Encoder_Extendido := gEncoder_AbsolutoExtendido;
Encoder_Parada := gEncoder_OperativaB;
TeachingOperativaB := gEncoder_Absoluto - 40000;            //----- Valor que permite el inicio del teaching del encoder de parada -----//
Encoder_Extendido_OFFSET := 150;							//----- Valor para los casos de anomalia en que no detectamos inductivo de brazo extendido -----//
Encoder_Recogido_OFFSET := 150;								//----- Valor para los casos de anomalia en que no detectamos inductivo de brazo recogido -----//

Encoder_Parada_OFFSET := 200;								//----- Valor de OFFSET para la parada del brazo por encoder -----//

C40.NumID:=1;
C40.MatrizID[1]:=65;
C41.RespuestasTotales[1]:=16#1F;        					//----- Tiene que recibir informacion de 5 PDOs -----//

//-------------------------------------------------------------------------------------------//
//----------------------------Definicion temporizacion inicial-------------------------------//
//-------------------------------------------------------------------------------------------//
SEGUNDOS_ENCENDIDO := 10;
TIEMPO_CICLO_DESEADO := 15000;

//-------------------------------------------------------------------------------------------//
//----------------------------------------Anomalias------------------------------------------//
//-------------------------------------------------------------------------------------------//
//TIPO_ANOMALIA[0]  := 3;	
//----- Anomalias supervisor -----//
TIPO_ANOMALIA[1]  := 3;		
TIPO_ANOMALIA[2]  := 1;	

//----- Anomalias imágenes -----//
TIPO_ANOMALIA[3]  := 3;		
TIPO_ANOMALIA[4]  := 4;		
TIPO_ANOMALIA[5]  := 3;		
TIPO_ANOMALIA[6]  := 3;		
TIPO_ANOMALIA[7]  := 3;	
TIPO_ANOMALIA[8]  := 3;		
TIPO_ANOMALIA[9]  := 3;	

//----- Anomalías estados -----//
TIPO_ANOMALIA[10] := 1;		
TIPO_ANOMALIA[11] := 2;		
TIPO_ANOMALIA[12] := 2;		
TIPO_ANOMALIA[13] := 2;		
TIPO_ANOMALIA[14] := 2;		
TIPO_ANOMALIA[15] := 3;
TIPO_ANOMALIA[16] := 2;		
TIPO_ANOMALIA[17] := 0;	

//----- Anomalías secuencia carga -----//
TIPO_ANOMALIA[18] := 4;		
TIPO_ANOMALIA[19] := 1;		
TIPO_ANOMALIA[20] := 3;		
TIPO_ANOMALIA[21] := 2;		
TIPO_ANOMALIA[22] := 3;		
TIPO_ANOMALIA[23] := 3; 
TIPO_ANOMALIA[24] := 3;		
//TIPO_ANOMALIA[25] := 2;	

//----- Anomalías extensión -----//
TIPO_ANOMALIA[26] := 2;		 
TIPO_ANOMALIA[27] := 3;		
TIPO_ANOMALIA[28] := 2;		
TIPO_ANOMALIA[29] := 2;		
TIPO_ANOMALIA[30] := 2;		
TIPO_ANOMALIA[31] := 2; 

//----- Anomalías elevación -----//
TIPO_ANOMALIA[32] := 3;		
TIPO_ANOMALIA[33] := 2;		
TIPO_ANOMALIA[34] := 4;		
(*TIPO_ANOMALIA[35] := 2;		
TIPO_ANOMALIA[36] := 2;		
TIPO_ANOMALIA[37] := 2;		
TIPO_ANOMALIA[38] := 2;		
TIPO_ANOMALIA[39] := 2; *)

END_PROGRAM

// StandardPLC/Application/CÓDIGO/SUPERVISOR
PROGRAM SUPERVISOR
VAR CONSTANT
	TOTALANOMALIAS 			:INT := 39;
END_VAR
VAR
	estadoAnomalias	  		:ARRAY[0..TOTALANOMALIAS] OF BYTE;
	anomaliasEntrada 		:ARRAY[0..TOTALANOMALIAS] OF BOOL;
	rearme 					:BOOL;
	estadoManual 			:BOOL;
	A_EstadoReposo 			:BOOL;

	mensajeAnomalia 		:BYTE;
	controlEstados 			:BYTE;

	(*Auxiliares*)
	i 						:INT;
	j 						:INT;
END_VAR
VAR_OUTPUT
END_VAR

(*//////////////////////////////////////////////////////////////////////////////////////////////////////////////////////////////////////////////////////////////////////////////////////////////////////////////////////////////////////////////////
SUPERVISOR (PRG)                     

Description:	Las anomalias son administradas en este modulo.
				Existen 4 estados distintos de anomalia (variable estadoAnomalias):
					0: Activa
					1: desactivada
					2: pausa
					3: seguro
				Para cada anomalia, tenemos 5 valores de severidad:
					0: Advertencia autorearmable
					1: Advertencia rearmable
					2: Severa (E-Frame a estado seguro)
					3: Crítica (rearmable con seta)
					4: Fatal (no rearmable)
				
				Cuando no tenemos anomalia, el valor es 1. Siempre que es detectada una anomalia, el valor es cambiado para 0

////////////////////////////////////////////////////////////////////////////////////////////////////////////////////////////////////////////////////////////////////////////////////////////////////////////////////////////////////////////////////*)

//-------------------------------------------------------------------------------------------//
//-------------------------Hacer reset a la variable estadoAnomalias-------------------------//
//-------------------------------------------------------------------------------------------//
IF PrimerCiclo THEN
	TIPO_ANOMALIA[1] := 3;									//----- Anomalía cadena seguridad -----//
	FOR i:=0 TO TOTALANOMALIAS DO 
		estadoAnomalias[i] := 1;            				//----- Para todas las anomalias contempladas en la PARAMETRIZACION, el estado de anomalia es iniciado como anomalia desactivada -----//
	END_FOR;
END_IF;

IF gFinEncendido THEN
	
	anomaliasEntrada 	:= gSupE_AnomaliasEntrada;
	rearme 				:= gEntradasPLC.BotonRearme;       
	estadoManual 		:= (gEstadoEframe=Manual) OR (gEstadoEframe=Automatico); 
	A_EstadoReposo 		:= ((gEstadoCarga=cargado) OR (gEstadoCarga=descargado));
	
	//----------------------- estadoAnomalias para la cadena de seguridad -------------------------//
	IF (NOT anomaliasEntrada[1]) THEN
		estadoAnomalias[1] := 0;
	ELSIF ( (estadoAnomalias[1]=0) AND anomaliasEntrada[1] ) THEN
		estadoAnomalias[1] := 3;
	ELSIF ( (estadoAnomalias[1]=3) AND rearme ) THEN    			//----- Si tenemos anomalia en la seta -----//
		IF A_EstadoReposo THEN      								//----- y tenemos en E-Frame cargado o descargado -----//
			estadoAnomalias[1] := 1;     							//----- pasamos el estado de la anomalia como siendo una advertencia autorearmable activa -----//
		ELSE 
			estadoAnomalias[1] := 2;     							//----- si no , tenemos una anomalia severa -----//
		END_IF;
	ELSIF ( (estadoAnomalias[1]=2) AND estadoManual ) THEN     		//----- tenemos una anomalia severa en la cadena de seguridad y estamos en modo manual -----//
		estadoAnomalias[1] := 1;                               		//----- pasamos el estado de la anomalia para una advertencia autorearmable activa -----//
	END_IF;

	//----------------------------------Cambiar estadoAnomalias----------------------------------//
	FOR i:=1 TO (TOTALANOMALIAS-1) DO
		CASE TIPO_ANOMALIA[i] OF
			0: // Advertencia autorearmable. Cuando desaparece origen anomalía. 0:ACTIVA, 1:DESACTIVADA
				estadoAnomalias[i] := BOOL_TO_BYTE(anomaliasEntrada[i]);
			1: // Advertencia rearmable  . Limpiamos anomalía con REARMAR. 0:ACTIVA, 1:DESACTIVADA
				IF (NOT anomaliasEntrada[i]) THEN     				//----- Si tenemos una anomalia, cambiamos su estado para ACTIVO -----//
					estadoAnomalias[i] := 0;
				END_IF;
				IF ( rearme ) THEN    								//----- Así que pulsemos rearme, desactivamos la variable de anomalia -----//
					estadoAnomalias[i] := 1; 
				END_IF;
			2: // Severa - a estado seguro. Permite pausar anomalía con REARMAR, pero desaparece cuando entramos en degradado/manual para corrección.
			    // 0:ACTIVA, 1:DESACTIVADA, 2:PAUSA
				IF ( (estadoAnomalias[i]=1) AND (NOT anomaliasEntrada[i]) ) THEN     //----- Si la variable de anomalia esta desactiva y tenemos una anomalia, pasamos la variable para el estado ACTIVO -----//
					estadoAnomalias[i] := 0;
				ELSIF ( (estadoAnomalias[i]=0) AND rearme ) THEN     //----- Si la variable de anomalia esta en estado activo y pulsamos rearme, ponemos su estado como sendo PAUSA -----//
					estadoAnomalias[i] := 2;
				ELSIF ( ((estadoAnomalias[i]=2) OR (estadoAnomalias[i]=0)) AND rearme ) THEN    //----- Si tenemos el estado de la variable como PAUSA o ACTIVA y cambiamos a modo manual, quitamos anomalia -----//
					estadoAnomalias[i] := 1;
				END_IF;
			3: // Crítica - rearmable con seta . Requieren reset por parte de cadena de seguridad. 0:ACTIVA, 1:DESACTIVADA
				gSalidasPLC.LuzBotonRearme := TOF_Rearme.Q;
				IF rearme THEN        //----- Si cargamos el boton rearme, quitamos la anomalia. Si no, si continuamos con anomalia, la variable estadoAnomalias continua con anomalia activa -----//
					estadoAnomalias[i] := 1;
					gSalidasPLC.LuzBotonRearme := FALSE;
				ELSIF (NOT anomaliasEntrada[i]) THEN
					estadoAnomalias[i] := 0;
				END_IF;
			4: // Fatal - no rearmable. Podemos pausar con cadena de seguridad, pero no se rearmarán. 0:ACTIVA, 1:DESACTIVADA, 2:PAUSA
				IF ( (estadoAnomalias[i]=1) AND (NOT anomaliasEntrada[i]) ) THEN    //----- Si la variable esta DESACTIVA y tenemos una anomalia, cambiamos el estado de la variable para ACTIVA -----//
					estadoAnomalias[i] := 0;
				ELSIF ( (estadoAnomalias[i]=0) AND rearme ) THEN     //----- Si la variables de las anomalias esta ACTIVA y pulsamos rearme, cambiamos su estado para PAUSA	-----//
					estadoAnomalias[i] := 2;
				END_IF;
		END_CASE;
	END_FOR;

	//----- Si tenemos anomalias en extension, reset respectivo módulo control -----//
	gSupS_ResetExtension :=0;

	FOR i:=26 TO 31 DO					
		IF (anomaliasEntrada[i]=0) AND (NOT LASER_AUX) THEN     //----- Si tenemos alguna anomalia -----//
			gSupS_ResetExtension :=1;       					//----- Pasa la variable a 1. Desencadea anomalia en el brazo -----//
			EXIT; 
		END_IF; 	
	END_FOR;
	
	controlEstados 		:= 0;
	mensajeAnomalia 	:= 0;
	
	//----- De acuerdo con el tipo de anomalia que tenemos, vamos escribir la variable mensajeAnomalia para enviar al AGV -----//
	IF ( estadoAnomalias[1]=0 ) THEN   				//----- Anomalia cadena de seguridad -----//
		mensajeAnomalia := 1;	
		controlEstados := 6;
	ELSIF ( estadoAnomalias[1]=3 ) THEN     		//----- Cadena de seguridad en estado seguro -----//
		mensajeAnomalia := 2;	
		controlEstados := 4;
	ELSE
		FOR j:=4 TO 0 BY (-1) DO                   //----- De más a menos severidad -----//
			FOR i:=3 TO (TOTALANOMALIAS-1) DO      //----- Todas las anomalías -----//
				IF ( TIPO_ANOMALIA[i]=j) AND (estadoAnomalias[i]<>1 ) THEN      //----- Si para i tenemos la anomalia j y la variable de anomalia esta en un caso distinto de DESACTIVO -----//
					mensajeAnomalia := INT_TO_BYTE(i);
					CASE j OF
						0: controlEstados := 1;
						1: controlEstados := 5;
						2: 	IF estadoAnomalias[i]=0 THEN 
								controlEstados := 3; 
							ELSE controlEstados := 2;    //----- Si hemos quitado la seta, entra en el seguiente estado de anomalia que es el 3 (necesario llevar E-Frame a posicion inicial) -----//
								mensajeAnomalia := 3; 
							END_IF;
						3: 	IF estadoAnomalias[i]=0 THEN 
								controlEstados := 6; 
							ELSE 
								controlEstados := 2; 
								mensajeAnomalia := 2; //3
							END_IF;
						4: 	IF estadoAnomalias[i]=0 THEN 
								controlEstados := 6; 
							ELSE 
								controlEstados := 4; 
							END_IF;
					END_CASE;
					EXIT;
				END_IF;
			END_FOR;

			IF ( mensajeAnomalia<>0 ) THEN		//----- Si tenemos valor en la variable mensajeAnomalia, tenemos anomalia -----//
				EXIT;
			END_IF;

		END_FOR;
	END_IF;

	gSupS_MensajeAnom 		:= mensajeAnomalia;
	gSupS_ControlEstados 	:= controlEstados;
END_IF;

END_PROGRAM

// StandardPLC/Application/CÓDIGO/ESTADOS
	PROGRAM ESTADOS
VAR
	OrdenDegradado			:BOOL;
	OrdenManual				:BOOL;
	OrdenAuto				:BOOL;
	FrenteAestacion			:BOOL;

	TON_SalirManual			:TON;
	
	Tempo_Actual 			:TIME;
	RetenerEstado			:EstadoEframe;
	CondicionReinicio		:BOOL;
	EstadoAnomaliaA			:BYTE;

	AnomaliaIndeterminado 	:BOOL;
	TON_Posicionado 		:TON;
	AnomaliaPartida 		:BOOL;
	TON_AnomaliaReinicio	:TON;
	AnomaliaReinicio		:BOOL;
END_VAR
VAR_OUTPUT
END_VAR

(*//////////////////////////////////////////////////////////////////////////////////////////////////////////////////////////////////////////////////////////////////////////////////////////////////////////////////////////////////////////////////
ESTADOS (PRG)                     

Description:  Máquina estados principal e-frame. Tenemos 7 estados:

				Identificar 	-> Condiciones arranque. Identifica estado seguro.
				Reposo			-> Brazo retraído, sin orden de carga o descarga.
				Automatico		-> E-Frame ejecutando operativa em modo automatico.
				Degradado		-> Control del brazo con auxilio de un taladro. Salidas del PLC desactivas.
				Manual			-> Control del E-Frame por botones (movimiento del brazo y movimiento de las levas). 
								En este modo, no tenemos anomalias.
				Reinicio		-> Estado utilizado para cuando salimos del modo manual o degradado.
				Anomalía		-> Fueron detetadas anomalias en el funcionamiento.

/////////////////////////////////////////////////////////////////////////////////////////////////////////////////////////////////////////////////////////////////////////////////////////////////////////////////////////////////////////////////////*)

IF gFinEncendido THEN
	//-------------------------------------------------------------------------------------------//
	//-----------CASE para el control del estado de la carga cuando iniciamos E-Frame------------//
	//-------------------------------------------------------------------------------------------//
	IF (gCargaOPT = indeterminado) AND gEntradasPLC.ModoAutomatico THEN
		PalabraAnomalia.2 := 0;
	ELSE
		PalabraAnomalia.2 := 1;
	END_IF
	
	IF (NOT gEntradasPlc.InductivoSubirLevas) AND gEntradasPlc.InductivoBajarLevas  THEN  
		 gCargaOPT := 2;
	ELSIF  gEntradasPlc.InductivoSubirLevas AND (NOT gEntradasPlc.InductivoBajarLevas)  THEN     
		 gCargaOPT := 1; 
	ELSIF (TON_BajarLevas.Q AND (NOT gEntradasPlc.InductivoBajarLevas))  OR (TON_SubirLevas.Q AND (NOT gEntradasPlc.InductivoSubirLevas)) THEN
		gCargaOPT := 3;
	END_IF
	
	CASE gCargaOPT OF
		1:  // E-Frame cargado
			gEstadoCarga := cargado;

		2:  // E-Frame descargado
			gEstadoCarga := descargado;
			
		3:  // E-Frame con estado de carga indeterminado. Si el estado de la carga es indeterminado, generamos anomalia
			gEstadoCarga := indeterminado;
	END_CASE	

	OrdenDegradado 		:= (NOT gEntradasPLC.Modo_Degradado);
	OrdenManual 		:= (NOT gEntradasPLC.ModoAutomatico);
	OrdenAuto			:= gEntradasPLC.ModoAutomatico AND (gEntradasAGV.OrdenCarga OR gEntradasAGV.OrdenDescarga OR (gEntradasAGV.OrdenDescarga AND gEntradasAGV.OrdenDescargaB));
	FrenteAestacion 	:= gEntradasPLC.ParadaPrecisaEFrame;
	
	IF ( OrdenDegradado AND (gSupS_ControlEstados=0 OR gSupS_ControlEstados=2) AND (NOT gEntradasPLC.Manual_ExtenderBrazo) ) OR
 	   ( OrdenDegradado AND (gSupS_ControlEstados=0 OR gSupS_ControlEstados=2) AND gEntradasPLC.Manual_ExtenderBrazo)THEN
		gEstadoEframe := Degradado;
		OPT := indeterminado_OPT;
	ELSIF ( OrdenManual AND (gSupS_ControlEstados=0 OR gSupS_ControlEstados=2) ) THEN
		gEstadoEframe := Manual;
	ELSIF ( gSupS_ControlEstados <>0 ) THEN 
		gEstadoEframe := Anomalia;
	END_IF;	

//-------------------------------------------------------------------------------------------//
//-------Cambia los estados del E-Frame teniendo en cuenta los valores de la sensorica-------//
//-------------------------------------------------------------------------------------------//
	CASE gEstadoEframe OF
		Identificar:
			AnomaliaPartida := FALSE;
			AnomaliaIndeterminado := FALSE;
			IF ( (NOT OrdenAuto) AND gEntradasPLC.InductivoBrazoRec ) THEN    
				IF ( gEstadoCarga=cargado ) THEN
					gEstadoEframe := Reposo;
				ELSIF ( gEstadoCarga=descargado ) THEN
					gEstadoEframe := Reposo;
				ELSIF ( gEstadoCarga=indeterminado ) THEN
					AnomaliaIndeterminado := TRUE;
				ELSE
					AnomaliaPartida := TRUE;
				END_IF;
				gEframeConCarga := (gEntradasPLC.DeteccionCarga1 AND gEntradasPLC.DeteccionCarga2);      
			END_IF;

		Reposo:
			AccionBrazo := A_Parar;
			gSalidasPLC.LuzBotonRearme := FALSE;
			TON_SalirManual( IN:=FALSE);
			IF ( ((gEstadoCarga=cargado AND gEntradasAGV.OrdenDescarga AND FrenteAestacion) OR (gEstadoCarga=cargado AND gEntradasAGV.OrdenDescarga AND gEntradasAGV.OrdenDescargaB) OR 
			  (gEstadoCarga=descargado AND gEntradasAGV.OrdenCarga AND FrenteAestacion))  AND gEntradasAGV.Habilitar AND (CondicionReinicio = 0) ) THEN
				gEstadoEframe := Automatico;
			ELSIF (gEstadoCarga=cargado AND (NOT gEntradasPlc.InductivoSubirLevas) AND (NOT gEntradasPLC.DeteccionCarga1) AND (NOT gEntradasPLC.DeteccionCarga2)) OR 
				(gEstadoCarga=descargado AND (NOT gEntradasPlc.InductivoBajarLevas) AND gEntradasPLC.DeteccionCarga1 AND gEntradasPLC.DeteccionCarga2) THEN
				gSupE_AnomaliasEntrada[34] := 0;
			END_IF;
			RetenerEstado := Reposo;
	
		Automatico:
			gSalidasPLC.LuzBotonRearme := FALSE;
			IF ((gEstadoCarga=cargado OR gEstadoCarga=descargado) AND (NOT OrdenAuto) AND (CondicionReinicio = 0) AND gEntradasPLC.InductivoBrazoRec) THEN //OR (gEstadoCarga=cargado AND (NOT gEntradasAGV.OrdenDescarga) AND (CondicionReinicio =0)) OR (gEstadoCarga=descargado AND (NOT gEntradasAGV.OrdenCarga) AND (CondicionReinicio =0)) ) 
				gEstadoEframe := Reposo;
			END_IF;
			RetenerEstado := Automatico;
			
		Degradado:           //----- Cuando dejamos el modo degradado y le damos el rearme, el estado del E-Frame se pasa para el modo de reinicio -----//
			CondicionReinicio := 1;

		Manual:
			IF (NOT OrdenManual) THEN
				gSalidasPLC.LuzBotonRearme := TOF_Rearme.Q;
			ELSE
				gSalidasPLC.LuzBotonRearme := FALSE;
			END_IF
			
			CondicionReinicio := 1;
			IF ( TON_SalirManual.Q ) THEN   //----- Cuando dejamos el modo manual y le damos el rearme, el estado del E-Frame se pasa para el modo de reinicio -----//
				gEstadoEframe := Reinicio;
				gSalidasPLC.LuzBotonRearme := FALSE;
				AnomaliaReinicio := 0;
			END_IF;
			RetenerEstado := Manual;
	
		Reinicio:
			AnomaliaReinicio := 0;
			IF CondicionReinicio THEN
				CondicionReinicio := 0;
			END_IF;
			IF ( gDispS_ExtensionEstado<>1 ) THEN
				AnomaliaReinicio := 1;
			ELSIF ( (gEstadoCarga=cargado) OR (gEstadoCarga=descargado) ) THEN
				gEstadoEframe := Reposo;
			END_IF;
			RetenerEstado := Reinicio;
	
		Anomalia:
			IF ( ((EstadoAnomaliaA=1) OR (EstadoAnomaliaA=5)) AND (gSupS_ControlEstados=0) ) THEN     //----- Cuando dejamos de tener una anomalia, el E-Frame se vuelve al estado anterior -----//
				gEstadoEframe := RetenerEstado;
				EstadoAnomaliaA := 0;
			ELSIF ( ((gSupS_ControlEstados=1) OR (gSupS_ControlEstados=2) OR (gSupS_ControlEstados=3)) AND OrdenDegradado ) THEN    //----- Si tenemos una anomalia y estamos en modo degradado -----// 
				gEstadoEframe := Degradado;																							//----- el estado del E-Frame va a pasar para modo degradado -----//
				EstadoAnomaliaA := 0;    //----- En el modo degradado, se espera que el degradado sea desactidavo y que pulsemos el boton de rearme para que lo estado sea cambiado para reinicio -----//
				//----- Lo mismo pasa para MANUAL y REPOSO -----//
			ELSIF ( ((gSupS_ControlEstados=1) OR (gSupS_ControlEstados=2) OR (gSupS_ControlEstados=3)) AND OrdenManual ) THEN
				gEstadoEframe := Manual;
				EstadoAnomaliaA := 0;
			ELSIF ( ((EstadoAnomaliaA=4) OR (EstadoAnomaliaA=6) OR (EstadoAnomaliaA=0)) AND (gSupS_ControlEstados=0) ) THEN
				gEstadoEframe := Reposo;
				EstadoAnomaliaA := 0;
			ELSIF (EstadoAnomaliaA=0) AND (gSupS_ControlEstados=0) AND (NOT OrdenManual) THEN
				gEstadoEframe := Reposo;
			END_IF;

			EstadoAnomaliaA := gSupS_ControlEstados;
				
	END_CASE;
	
	TON_SalirManual( IN:=((NOT OrdenManual) AND gEntradasPLC.BotonRearme), PT:=T#2S, ET => Tempo_Actual  );      
	
	
//-------------------------------------------------------------------------------------------//
//-----------------------------------------Anomalias-----------------------------------------//
//-------------------------------------------------------------------------------------------//	
	//----- Anomalía por orden en reposo -----//
	IF ( (gEstadoEframe=Reposo) AND OrdenAuto AND (NOT FrenteAestacion) AND (gEntradasAGV.OrdenCarga OR (gEntradasAGV.OrdenDescarga AND (NOT gEntradasAGV.OrdenDescargaB))) ) THEN      
		gSupE_AnomaliasEntrada[10] := 0;
	ELSE
		gSupE_AnomaliasEntrada[10] := 1;
	END_IF;
	
	//----- No esta posicionado frente a la estacion -----//
	TON_Posicionado( IN:=(NOT FrenteAestacion), PT:=T#200MS );
	IF ( (gEstadoEframe=Automatico) AND TON_Posicionado.Q AND (NOT gEntradasAGV.OrdenDescargaB) ) THEN      //----- Se paso el tiempo y el E-Frame continua sin estar posicionado -----//
		gSupE_AnomaliasEntrada[11] := 0;                               //----- Es gerada anomalia -----//
	ELSE
		gSupE_AnomaliasEntrada[11] := 1;
	END_IF;
	
	//----- Anomalía identificando estado -----//
	IF ( (gEstadoEframe=Identificar) AND AnomaliaIndeterminado ) THEN
		gSupE_AnomaliasEntrada[12] := 0;
	ELSE
		gSupE_AnomaliasEntrada[12] := 1;
	END_IF;
	
	//----- Anomalia estado inaceptable en reposo: estado del e-frame en reposo y brazo en posicion distinta de recogido -----//
	IF ( (gEstadoEframe=Reposo) AND (gDispS_ExtensionEstado<>1) ) OR 			
       ((gEstadoEframe=Identificar) AND (NOT OrdenAuto) AND (NOT gEntradasPLC.InductivoBrazoRec)) OR 
       ((gEstadoEframe=Identificar) AND OrdenAuto AND (NOT gEntradasPLC.InductivoBrazoRec)) THEN
		gSupE_AnomaliasEntrada[13] := 0;
	ELSE
		gSupE_AnomaliasEntrada[13] := 1;
	END_IF;
	
	//----- Anomalia estado de partida -----//
	IF ( (gEstadoEframe=Identificar) AND AnomaliaPartida ) THEN
		gSupE_AnomaliasEntrada[14] := 0;
	ELSE
		gSupE_AnomaliasEntrada[14] := 1;
	END_IF;
	
	// Anomalia estado inaceptable con convoy en marcha
	(*IF ( (gEstadoEframe<>Reposo) AND (NOT gEntradasAGV.Habilitar) AND ((COMUNICACION_CAN.O_EstadoCAN AND 16#0F)<>16#0F) ) THEN
		gSupE_AnomaliasEntrada[15] := 0;
	ELSE
		gSupE_AnomaliasEntrada[15] := 1;
	END_IF;*)
	
	//----- Anomalia posición inaceptable reinicio -----//
	TON_AnomaliaReinicio( IN:=AnomaliaReinicio, PT:=T#200MS);           //----- AnomaliaReinicio: cuando estamos en estado de reposo pero el brazo no esta recogido -----//
	IF ( (gEstadoEframe=Reinicio) AND TON_AnomaliaReinicio.Q ) THEN
		gSupE_AnomaliasEntrada[16] := 0;
	ELSE
		gSupE_AnomaliasEntrada[16] := 1;
		AnomaliaReinicio := FALSE;
	END_IF;
	
	//----- Anomalía detección láser en automático -----//
	IF ( LASER_AUX ) THEN 
		gSupE_AnomaliasEntrada[17] := 0; 
	ELSE
		gSupE_AnomaliasEntrada[17] := 1;
	END_IF;
END_IF;

END_PROGRAM

// StandardPLC/Application/CÓDIGO/AUX_IFM/fb_OutputGroupAddConf_sp_ST_V02
FUNCTION_BLOCK fb_OutputGroupAddConf_sp_ST_V02
VAR_INPUT
	IN_ResetError:BOOL;	
	IN_uiChannel:UINT;
	IN_eModeChannel:ifmOutGroup.MODE_OUTPUT_GROUP;	
	IN_eDestination:ifmIOconfigDiagProt.DEST;
	IN_eDiagMode:ifmIOconfigDiagProt.eDIAG_PROT_MODE;
	IN_DetectionTime:UINT;
	IN_DiagLimMin:UINT;
	IN_DiagLimMax:UINT;

	IN_Value:BOOL;
	
		
END_VAR
	
VAR_OUTPUT
	OUT_Done:BOOL;
	OUT_Error:BOOL;
	OUT_DiagInfo:ifmTypes.DIAG_INFO;	
	OUT_DiagInfoProt: ifmTypes.DIAG_INFO;
	OUT_DiagInfoLevel: ifmTypes.DIAG_INFO;	
END_VAR
VAR
	
	l_xExecute:BOOL;
	ConfigDiagLevel: ifmIOconfigDiagProt.ConfigDiagLevel;
	ConfigDiagProt: ifmIOconfigDiagProt.ConfigDiagProt;

	l_xExecute_DiagLevel:BOOL;
	l_xExecuted_DiagLevel:BOOL;	
	l_xExecute_DiagProt:BOOL;
	l_xExecuted_DiagProt:BOOL;
	R_TRIG_Execute: R_TRIG;
	OutputGroup:ifmOutGroup.OutputGroup;
	R_TRIG_Done: R_TRIG;
END_VAR
VAR // added by the converter: edge detectors and wires of the graphical bodies
    _w1 : BOOL;
END_VAR

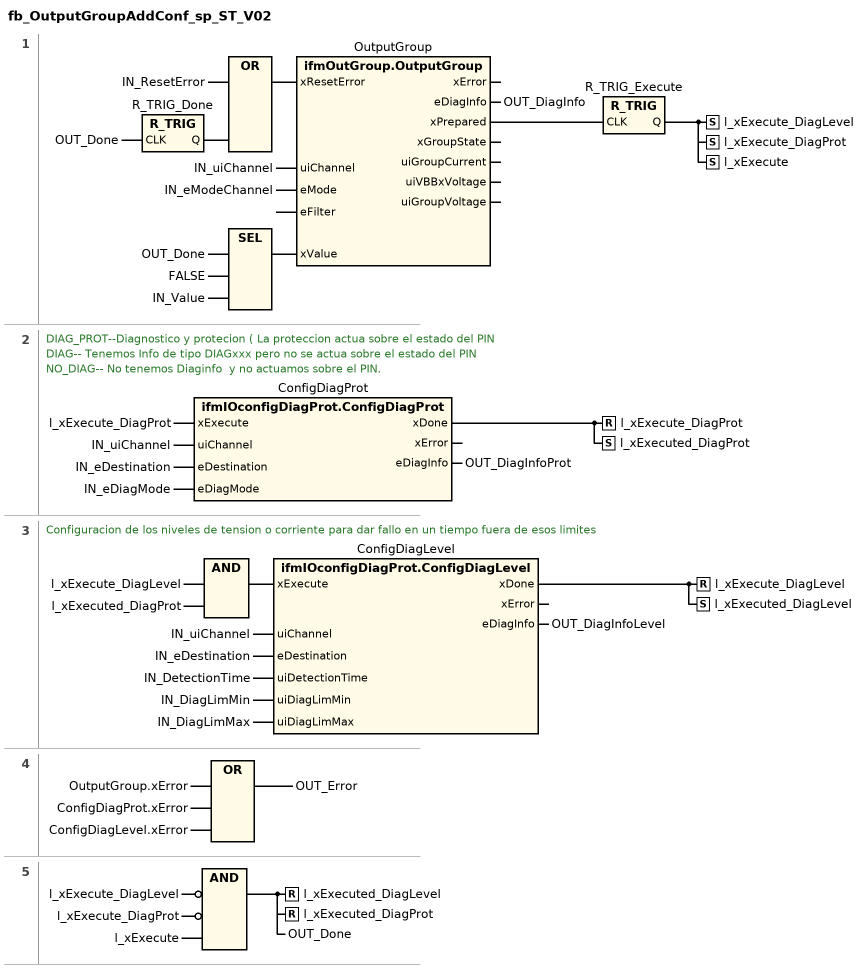
// NETWORK 1
R_TRIG_Done(CLK := OUT_Done); // R_TRIG
OutputGroup(
    xResetError := IN_ResetError OR R_TRIG_Done.Q,
    uiChannel := IN_uiChannel,
    eMode := IN_eModeChannel,
    xValue := SEL(OUT_Done, FALSE, IN_Value),
    eDiagInfo => OUT_DiagInfo); // ifmOutGroup.OutputGroup
R_TRIG_Execute(CLK := OutputGroup.xPrepared); // R_TRIG
l_xExecute_DiagLevel S= R_TRIG_Execute.Q;
l_xExecute_DiagProt S= R_TRIG_Execute.Q;
l_xExecute S= R_TRIG_Execute.Q;

// NETWORK 2
// DIAG_PROT--Diagnostico y protecion ( La proteccion actua sobre el estado del PIN
// DIAG-- Tenemos Info de tipo DIAGxxx pero no se actua sobre el estado del PIN
// NO_DIAG-- No tenemos Diaginfo  y no actuamos sobre el PIN.
ConfigDiagProt(
    xExecute := l_xExecute_DiagProt,
    uiChannel := IN_uiChannel,
    eDestination := IN_eDestination,
    eDiagMode := IN_eDiagMode,
    eDiagInfo => OUT_DiagInfoProt); // ifmIOconfigDiagProt.ConfigDiagProt
l_xExecute_DiagProt R= ConfigDiagProt.xDone;
l_xExecuted_DiagProt S= ConfigDiagProt.xDone;

// NETWORK 3
// Configuracion de los niveles de tension o corriente para dar fallo en un tiempo fuera de esos limites
ConfigDiagLevel(
    xExecute := l_xExecute_DiagLevel AND l_xExecuted_DiagProt,
    uiChannel := IN_uiChannel,
    eDestination := IN_eDestination,
    uiDetectionTime := IN_DetectionTime,
    uiDiagLimMin := IN_DiagLimMin,
    uiDiagLimMax := IN_DiagLimMax,
    eDiagInfo => OUT_DiagInfoLevel); // ifmIOconfigDiagProt.ConfigDiagLevel
l_xExecute_DiagLevel R= ConfigDiagLevel.xDone;
l_xExecuted_DiagLevel S= ConfigDiagLevel.xDone;

// NETWORK 4
OUT_Error := OutputGroup.xError OR ConfigDiagProt.xError OR ConfigDiagLevel.xError;

// NETWORK 5
_w1 := NOT l_xExecute_DiagLevel AND NOT l_xExecute_DiagProt AND l_xExecute;
l_xExecuted_DiagLevel R= _w1;
l_xExecuted_DiagProt R= _w1;
OUT_Done := _w1;

END_FUNCTION_BLOCK

// StandardPLC/Application/CÓDIGO/AUX_IFM/fb_OutputAddConf_sp_ST_V02
FUNCTION_BLOCK fb_OutputAddConf_sp_ST_V02
VAR_INPUT
	IN_ResetError:BOOL;	
	IN_uiChannel:UINT;
	IN_eModeChannel:ifmIOcommon.MODE_OUTPUT;	
	IN_eDestination:ifmIOconfigDiagProt.DEST;
	IN_eDiagMode:ifmIOconfigDiagProt.eDIAG_PROT_MODE;
	IN_DetectionTime:UINT;
	IN_DiagLimMin:UINT;
	IN_DiagLimMax:UINT;

	IN_Value:BOOL;
	
		
END_VAR
	
VAR_OUTPUT
	OUT_Done:BOOL;
	OUT_Error:BOOL;
	OUT_DiagInfo:ifmTypes.DIAG_INFO;	
	OUT_DiagInfoProt: ifmTypes.DIAG_INFO;
	OUT_DiagInfoLevel: ifmTypes.DIAG_INFO;	
END_VAR
VAR
	
	l_xExecute:BOOL;
	ConfigDiagLevel: ifmIOconfigDiagProt.ConfigDiagLevel;
	ConfigDiagProt: ifmIOconfigDiagProt.ConfigDiagProt;

	l_xExecute_DiagLevel:BOOL;
	l_xExecuted_DiagLevel:BOOL;	
	l_xExecute_DiagProt:BOOL;
	l_xExecuted_DiagProt:BOOL;
	R_TRIG_Execute: R_TRIG;
	Output:ifmIOcommon.Output;
	R_TRIG_Done: R_TRIG;
END_VAR
VAR // added by the converter: edge detectors and wires of the graphical bodies
    _w1 : BOOL;
END_VAR

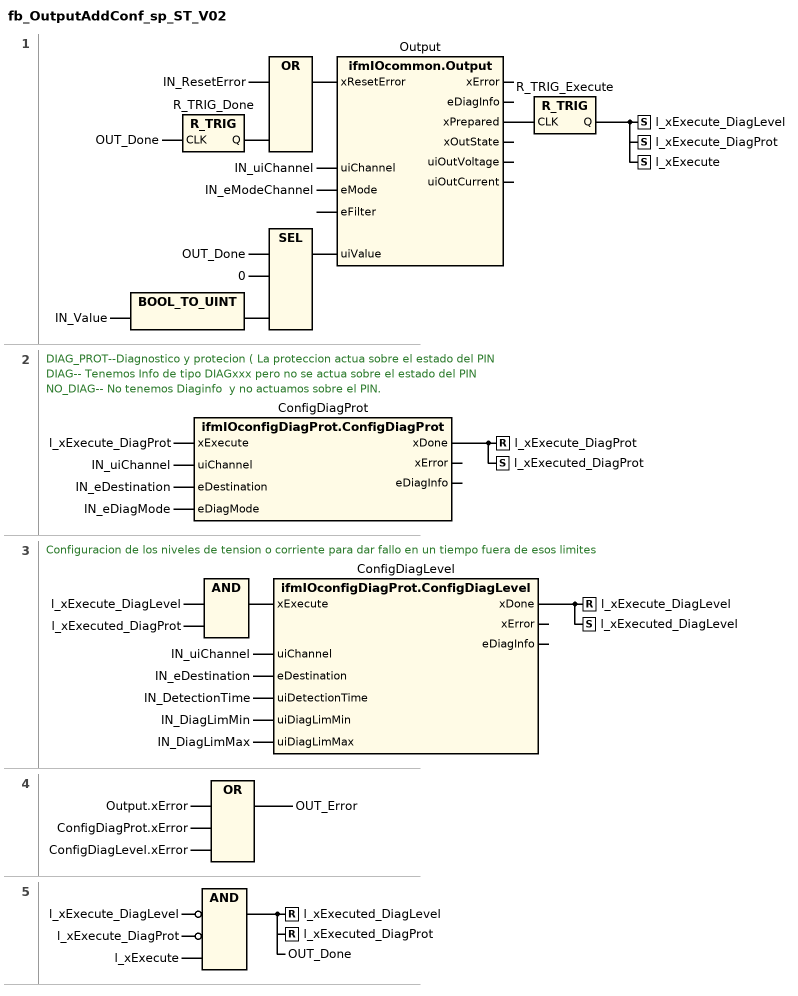
// NETWORK 1
R_TRIG_Done(CLK := OUT_Done); // R_TRIG
Output(
    xResetError := IN_ResetError OR R_TRIG_Done.Q,
    uiChannel := IN_uiChannel,
    eMode := IN_eModeChannel,
    uiValue := SEL(OUT_Done, 0, BOOL_TO_UINT(IN_Value))); // ifmIOcommon.Output
R_TRIG_Execute(CLK := Output.xPrepared); // R_TRIG
l_xExecute_DiagLevel S= R_TRIG_Execute.Q;
l_xExecute_DiagProt S= R_TRIG_Execute.Q;
l_xExecute S= R_TRIG_Execute.Q;

// NETWORK 2
// DIAG_PROT--Diagnostico y protecion ( La proteccion actua sobre el estado del PIN
// DIAG-- Tenemos Info de tipo DIAGxxx pero no se actua sobre el estado del PIN
// NO_DIAG-- No tenemos Diaginfo  y no actuamos sobre el PIN.
ConfigDiagProt(
    xExecute := l_xExecute_DiagProt,
    uiChannel := IN_uiChannel,
    eDestination := IN_eDestination,
    eDiagMode := IN_eDiagMode); // ifmIOconfigDiagProt.ConfigDiagProt
l_xExecute_DiagProt R= ConfigDiagProt.xDone;
l_xExecuted_DiagProt S= ConfigDiagProt.xDone;

// NETWORK 3
// Configuracion de los niveles de tension o corriente para dar fallo en un tiempo fuera de esos limites
ConfigDiagLevel(
    xExecute := l_xExecute_DiagLevel AND l_xExecuted_DiagProt,
    uiChannel := IN_uiChannel,
    eDestination := IN_eDestination,
    uiDetectionTime := IN_DetectionTime,
    uiDiagLimMin := IN_DiagLimMin,
    uiDiagLimMax := IN_DiagLimMax); // ifmIOconfigDiagProt.ConfigDiagLevel
l_xExecute_DiagLevel R= ConfigDiagLevel.xDone;
l_xExecuted_DiagLevel S= ConfigDiagLevel.xDone;

// NETWORK 4
OUT_Error := Output.xError OR ConfigDiagProt.xError OR ConfigDiagLevel.xError;

// NETWORK 5
_w1 := NOT l_xExecute_DiagLevel AND NOT l_xExecute_DiagProt AND l_xExecute;
l_xExecuted_DiagLevel R= _w1;
l_xExecuted_DiagProt R= _w1;
OUT_Done := _w1;

END_FUNCTION_BLOCK

// StandardPLC/Application/CÓDIGO/IMAGENES
PROGRAM IMAGENES
VAR
	EntradaCodificada		:BYTE;
	PosicionGrupoA			:BYTE;
	ByteInicial				:BYTE;
END_VAR
VAR_OUTPUT
END_VAR

(*/////////////////////////////////////////////////////////////////////////////////////////////////////////////////////////////////////////////////////////////////////////////////////////////////////////////////////////////////////////////////
IMAGENES (PRG)                     

Description:  Identificacion de las entradas del PLC. 
			  Comunicacion CAN con el AGV (Identificacion del numero del E-Frame y rececion de informacion por parte del AGV. 
///////////////////////////////////////////////////////////////////////////////////////////////////////////////////////////////////////////////////////////////////////////////////////////////////////////////////////////////////////////////////// *)

//-------------------------------------------------------------------------------------------//
//------------------------------Definicion de las entradas PLC-------------------------------//
//-------------------------------------------------------------------------------------------//
IN01_WIRED_INPUTS();

//-------------------------------------------------------------------------------------------//
//-------------------------Asignación de las entradas fisicas del PLC------------------------//
//-------------------------------------------------------------------------------------------//
EntradaCodificada.0					:= E.4;			//----- Entrada 63: AGV 1 -----//
EntradaCodificada.1                 := E.5;		    //----- Entrada 64: AGV 2 -----//
EntradaCodificada.2                 := E.6;		    //----- Entrada 65: AGV 3 -----//
EntradaCodificada.3                 := E.7;		    //----- Entrada 66: AGV 4 -----//
EntradaCodificada.4                 := E.8;		    //----- Entrada 67: AGV 5 -----//
EntradaCodificada.5                 := E.9;		    //----- Entrada 68: AGV 6 -----//

gEntradasPLC.Manual_ExtenderBrazo 	:= E2.4;		//----- Extender brazo manual -----//
gEntradasPLC.Manual_RecogerBrazo 	:= E2.5;		//----- Retrair brazo manual -----//

gEntradasPLC.Modo_Degradado 		:= E.11; 

gEntradasPLC.Manual_SubirLevas 		:= E.2;        
gEntradasPLC.Manual_BajarLevas		:= E.3;  

gEntradasPLC.ParadaPrecisaBrazo     := E.13;
gEntradasPLC.ParadaPrecisaEFrame	:=E.12;
 
gEntradasPLC.InductivoSubirLevas	:= E2.10;            
gEntradasPLC.InductivoBajarLevas    := E2.11; 
gEntradasPLC.DeteccionCarga1        := E2.14;
gEntradasPLC.DeteccionCarga2        := E2.15;
gEntradasPLC.DeteccionCargaExt      := E2.0;

gEntradasPLC.InductivoBrazoRec		:= E2.8;
gEntradasPLC.InductivoBrazoExt		:= E2.9;    

gEntradasPLC.SetaEmergenciaIN1		:= E2.6;
gEntradasPLC.SetaEmergenciaIN2		:= E2.7;

gEntradasPLC.Laser_OSSD1			:= E.0;
gEntradasPLC.Laser_OSSD2			:= E.1;

gEntradasPLC.BotonRearme 			:= E2.13;


//-------------------------------------------------------------------------------------------//
//-----------------------------Identificación del E-Frame a trabajar-------------------------//
//-------------------------------------------------------------------------------------------//
IF PrimerCiclo THEN
	CASE EntradaCodificada OF
		1:	PosicionGrupo := 1;
		2:	PosicionGrupo := 2;
		4:	PosicionGrupo := 3;
		8:	PosicionGrupo := 4;
		16:	PosicionGrupo := 5;
		32:	PosicionGrupo := 6;
		ELSE
			PosicionGrupo := 0;
	END_CASE;
	PosicionGrupoA := PosicionGrupo;

ELSE
	CASE EntradaCodificada OF
		1:	PosicionGrupoA := 1;
		2:	PosicionGrupoA := 2;
		4:	PosicionGrupoA := 3;
		8:	PosicionGrupoA := 4;
		16:	PosicionGrupoA := 5;
		32:	PosicionGrupoA := 6;
		ELSE
			PosicionGrupoA := 0;
	END_CASE;
END_IF;

//-------------------------------------------------------------------------------------------//
//----------------------------------Recepcion del dispositivo CAN----------------------------//
//-------------------------------------------------------------------------------------------//
COMUNICACION_CAN( I_OPERACION_CAN:=0 );

CASE PosicionGrupo OF
1: ByteInicial := 0;
2: ByteInicial := 2;
3: ByteInicial := 4;
4: ByteInicial := 6;
5: ByteInicial := 0;
6: ByteInicial := 2;
ELSE
	ByteInicial := 0;
END_CASE;

//-------------------------------------------------------------------------------------------//
//----------------------------------Asignacion entradas AGV----------------------------------//
//-------------------------------------------------------------------------------------------//
gEntradasAGV.Manual					:= COMUNICACION_CAN.O_MatrizRX_AGV[ByteInicial].0;
gEntradasAGV.Rearmar				:= COMUNICACION_CAN.O_MatrizRX_AGV[ByteInicial].1;
gEntradasAGV.EmergenciasAGV			:= COMUNICACION_CAN.O_MatrizRX_AGV[ByteInicial].2;
gEntradasAGV.Habilitar				:= COMUNICACION_CAN.O_MatrizRX_AGV[ByteInicial].3;           //----- Para nosotros, esto es convoy detenido -----//
gEntradasAGV.OrdenCarga				:= COMUNICACION_CAN.O_MatrizRX_AGV[ByteInicial].4;
gEntradasAGV.OrdenDescarga			:= COMUNICACION_CAN.O_MatrizRX_AGV[ByteInicial].5;
gEntradasAGV.ForzarBumper			:= COMUNICACION_CAN.O_MatrizRX_AGV[ByteInicial].6;
gEntradasAGV.OrdenDescargaB			:= COMUNICACION_CAN.O_MatrizRX_AGV[ByteInicial].7;

//-------------------------------------------------------------------------------------------//
//--------------------------------------Anomalias Imagenes-----------------------------------//
//-------------------------------------------------------------------------------------------//
IF gFinEncendido THEN       
	
	//----- Caída cadena seguridad -----//
	IF ( ((NOT gEntradasPLC.SetaEmergenciaIN1) AND (NOT gEntradasPLC.SetaEmergenciaIN2)) OR gEntradasAGV.EmergenciasAGV )THEN
		gSupE_AnomaliasEntrada[1] := 0;
	ELSE
		gSupE_AnomaliasEntrada[1] := 1;	
	END_IF

	//----- Anomalia identificación carro -----//
	IF ( (PosicionGrupo<>PosicionGrupoA) OR (PosicionGrupo=0) ) THEN	//----- No rearmable -----//
		gSupE_AnomaliasEntrada[4]:=FALSE;
	END_IF;

	//----- Anomalia comunicacion CAN -----//
	IF COMUNICACION_CAN.O_EstadoCAN.0 THEN   
		gSupE_AnomaliasEntrada[5] := 1;
	ELSE
		gSupE_AnomaliasEntrada[5] := 0;	
	END_IF
	
	IF COMUNICACION_CAN.O_EstadoCAN.1 THEN  
		gSupE_AnomaliasEntrada[7] := 1;
	ELSE
			gSupE_AnomaliasEntrada[7] := 0;
	END_IF
	
	
	//----- Anomalia comunicacion CAN con variador -----//
	IF C41.EstadoRX_Variador.0 THEN  
		gSupE_AnomaliasEntrada[6] := 1;
	ELSE
		gSupE_AnomaliasEntrada[6] := 0;
	END_IF
	
	//----- Variador con estado de anomalia -----//
	IF C41.Anomalia_Variador.0 THEN    
		gSupE_AnomaliasEntrada[8] := 1;
	ELSE
		gSupE_AnomaliasEntrada[8] :=  0;
	END_IF

	//----- Anomalias orden doble automático inaceptable -----//
	IF (gEntradasAGV.OrdenCarga AND gEntradasAGV.OrdenDescarga) OR (gEntradasAGV.OrdenCarga AND gEntradasAGV.OrdenDescargaB)
		OR (gEntradasAGV.OrdenCarga AND gEntradasAGV.OrdenDescarga AND gEntradasAGV.OrdenDescargaB) THEN
		gSupE_AnomaliasEntrada[9] := 0;
	ELSE
		gSupE_AnomaliasEntrada[9] := 1;
	END_IF;
END_IF;

END_PROGRAM

// StandardPLC/Application/CÓDIGO/Seguridades/Setas_Seguridad
PROGRAM Setas_Seguridad
VAR_INPUT
	IN_CanalA_Setas            :BOOL;
	IN_CanalB_Setas            :BOOL;
	
	IN_PulsadorRearme          :BOOL;
END_VAR
VAR
	SF_EQUIVALENT_SETAS        	:SF_EQUIVALENT;
	SF_EMERGENCYSTOP_SETAS     	:SF_EMERGENCYSTOP;
	
	TON_Led 					:TON;
	TOF_LED 					:TON;
	
	// Variables auxiliares
	S_LevasArribaDONE							:BOOL;
	S_LevasAbajoDONE							:BOOL;
	S_ParadaFotocelula							:BOOL;
	S_AUX_EFrameDescargado					    :BOOL;
	S_control_bajar								:INT;
	S_control_subir								:INT;
	S_Opt_Descarga								:INT;
	S_Opt_Descarga_ANT 							:INT;
	S_Opt_Descarga_B							:INT;
	S_Opt_DescargaB_ANT 						:INT;
	S_Opt_Carga									:INT;
	S_Opt_Carga_ANT 							:INT;
	S_AUX_CONT_Automatico						:INT;
	S_gVelocidad								:VelocidadPorTramo;
	S_gValorConsigna							:INT;
	S_gConsignaSalida							:INT;
	S_gEstadoRampa								:BOOL;
	S_gConsignaVariador							:INT;
	S_gConsignaA								:INT;
	S_gRampaTotal								:INT;
END_VAR

(*//////////////////////////////////////////////////////////////////////////////////////////////////////////////////////////////////////////////////////////////////////////////////////////////////////////////////////////////////////////////////
Setas_Seguridad (PRG)                     

Description:	Funcion de control de las setas
				
///////////////////////////////////////////////////////////////////////////////////////////////////////////////////////////////////////////////////////////////////////////////////////////////////////////////////////////////////////////////////// *)

OUT01_WIRED_OUTPUTS();

TON_Led( IN:=TOF_LED.Q, PT:=T#500MS);
TOF_LED( IN:=( NOT TON_Led.Q ), PT:=T#500MS);

IN_CanalA_Setas 	:= gEntradasPLC.SetaEmergenciaIN1;
IN_CanalB_Setas 	:= gEntradasPLC.SetaEmergenciaIN2;
IN_PulsadorRearme 	:= gEntradasPLC.BotonRearme;

SF_EQUIVALENT_SETAS(Activate:=TRUE, S_CHANNELA:=gEntradasPLC.SetaEmergenciaIN1,S_CHANNELB:=gEntradasPLC.SetaEmergenciaIN2,DISCREPANCYTIME:=T#50MS);
SF_EMERGENCYSTOP_SETAS(Activate:=SF_EQUIVALENT_SETAS.Ready,S_ESTOPIN:=SF_EQUIVALENT_SETAS.S_EquivalentOut,S_STARTRESET:=0,S_AUTORESET:=0,RESET:=IN_PulsadorRearme);

CASE Setas_OPT OF	
	1:  // Espero en este estado que han pulsado seta en E-Frame o AGV
		IF (NOT SF_EMERGENCYSTOP_SETAS.S_ESTOPIN) OR gEntradasAGV.EmergenciasAGV THEN    
			Setas_OPT := 2;
		END_IF
		
		//----- Variables que indican si las levas han bajado o subido correctamente -----//
		S_LevasArribaDONE := LevasAbajoDONE;
		S_LevasAbajoDONE := LevasArribaDONE;
		S_ParadaFotocelula := ParadaFotocelula;
		S_AUX_EFrameDescargado := AUX_EFrameDescargado;
		S_control_bajar := control_bajar;
		S_control_subir := control_subir;
		S_Opt_Carga := Opt_Carga;
		S_Opt_Carga_ANT := Opt_Carga_ANT;
		S_Opt_Descarga := Opt_Descarga;
		S_Opt_Descarga_ANT := Opt_Descarga_ANT;
		S_Opt_Descarga_B := Opt_Descarga_B;
		S_Opt_DescargaB_ANT := Opt_DescargaB_ANT;
		S_AUX_CONT_Automatico := AUX_CONT_Automatico;
		S_gVelocidad := gVelocidad;
		S_gValorConsigna := gValorConsigna;	
		
		//----- Variables de SALIDAS() -----//
		S_gConsignaSalida := gConsignaSalida;
		S_gEstadoRampa := gEstadoRampa;
		S_gConsignaVariador := gConsignaVariador;
		S_gConsignaA := gConsignaA;
		S_gRampaTotal := gRampaTotal;
		

	2:  // He pulsado seta. Contactores abajo, contactor del variador abajo, channel rele de seguridad abajo, reseteo de todas las variables
		Laser := Bumper;
		SetaPulsada_AUX := TRUE;
		AccionBrazo := Setas_Parar;
		OPT := indeterminado_OPT;
		gSalidasPLC.Contactor := FALSE;
		gSalidasPLC.Contactor2 := FALSE;
		SS.1 := gSalidasPLC.Contactor;
		SS.10 := gSalidasPLC.Contactor2;
		gSalidasPLC.Ch1_ReleSeguridad := FALSE;
		gSalidasPLC.Ch2_ReleSeguridad := FALSE;
		gSalidasPLC.SubirLevas := FALSE;
		gSalidasPLC.BajarLevas := FALSE;
	
		//----- Reset de los timers de las levas -----//
		AUX_SubirLevas := FALSE;
		TON_SubirLevas(IN:=FALSE);
		AUX_BajarLevas := FALSE;
		TON_BajarLevas(IN:=FALSE);
		AUX_InitSubirLevas := FALSE;
		AUX_InitBajarLevas := FALSE;
		LevasAbajoDONE := FALSE;
		LevasArribaDONE := FALSE;
		ParadaFotocelula := FALSE;
		AUX_EFrameDescargado := FALSE;
		control_bajar := 1;
		control_subir := 1;
		Opt_Carga := 1;	
		Opt_Carga_ANT := 0;
		Opt_Descarga := 1;
		Opt_Descarga_ANT := 0;
		Opt_Descarga_B := 1;
		Opt_DescargaB_ANT := 0;
		AUX_CONT_Automatico := 0;
		AUX_DetecionCarga := FALSE;
		TON_DetecionCarga( IN:=FALSE);
		ACC02_ControlAutomatico.I_OrdenDescarga := FALSE;
		ACC02_ControlAutomatico.I_OrdenCarga := FALSE;
		ACC02_ControlAutomatico.I_OrdenDescargaB := FALSE;
		gVelocidad := SinConsigna;
		AccionBrazo_Laser := 0;
		ConsignaA := 0;
		RampaTotal := 0;

		IF SF_EMERGENCYSTOP_SETAS.S_ESTOPIN THEN
			Disp_SelectIndicadores := 14;
			gSalidasPLC.LuzBotonRearme := TOF_LED.Q;
			SS2.6 := gSalidasPLC.LuzBotonRearme;
		END_IF
		
		IF SF_EMERGENCYSTOP_SETAS.Reset THEN
			Setas_OPT := 3;
		END_IF
		
	3:  // Inicio del proceso de volver a habilitar todos los contactores y los channels
		RESET := TRUE;
		HabilitarVariador := TRUE;
		
		IF (SF_EMERGENCYSTOP_SETAS.S_ESTOPIN AND RESET AND SetaPulsada_AUX) THEN
			Setas_OPT := 4;
		END_IF
		
	4:  // Reset de las variables auxiliares y habilitacion de los channels del rele
		gSalidasPLC.LuzBotonRearme := FALSE;
		SS2.6 := gSalidasPLC.LuzBotonRearme;
		gSalidasPLC.Ch1_ReleSeguridad := TRUE;
		gSalidasPLC.Ch2_ReleSeguridad := TRUE;
		
		IF HabilitarVariador THEN
			gSalidasPLC.ContactorHabVariador := FALSE;
			AUX_TIMER := TRUE;
			TON_TIMER(IN:=AUX_TIMER,PT:=T#500MS);
	
			IF TON_TIMER.Q THEN
				gSalidasPLC.ContactorHabVariador := TRUE;
				C40.Estado_Init := 0;
				AUX_TIMER := FALSE;
				TON_TIMER(IN:=FALSE);
				Setas_OPT := 1;
				SetaPulsada_AUX := FALSE;
				RESET := FALSE;
				HabilitarVariador := FALSE;
				AUX_CONT_Automatico := 0;
			END_IF
		END_IF
END_CASE

END_PROGRAM

// StandardPLC/Application/CÓDIGO/Sub ACCIONES/ACC02_ControlAutomatico
PROGRAM ACC02_ControlAutomatico
VAR_INPUT
	I_OrdenCarga 					:BOOL;
	I_OrdenDescarga 				:BOOL;
	I_OrdenDescargaB				:BOOL;
	I_HABILITAR 					:BOOL;
END_VAR
VAR
	ControlExtension				:DISP01_CntrlExtensionGeneral_FB;
	Reposo_Automatico				:BOOL;
END_VAR

(*//////////////////////////////////////////////////////////////////////////////////////////////////////////////////////////////////////////////////////////////////////////////////////////////////////////////////////////////////////////////////
ACC02_ControlAutomatico (PRG)                      

Description:	Control automatico del E-Frame
				Existen 3 estados iniciales del E-Frame: init_descargado, init_cargado Y init_cargado_B
		 
///////////////////////////////////////////////////////////////////////////////////////////////////////////////////////////////////////////////////////////////////////////////////////////////////////////////////////////////////////////////////// *)

//-------------------------------------------------------------------------------------------//
//---------------------------------Anomalia por orden doble----------------------------------//
//-------------------------------------------------------------------------------------------//
IF (I_OrdenCarga AND I_OrdenDescarga AND (gEstadoEframe = Automatico)) OR (I_OrdenCarga AND I_OrdenDescargaB AND (gEstadoEframe = Automatico))
	OR (I_OrdenCarga AND I_OrdenDescarga AND I_OrdenDescargaB AND (gEstadoEframe = Automatico)) THEN 
	PalabraAnomalia.0 := 0; 
END_IF;

//-------------------------------------------------------------------------------------------//
//-----------------------Anomalia por no deteccion del encoder de hilo-----------------------//
//-------------------------------------------------------------------------------------------//
IF (Encoder = 0) THEN 
	PalabraAnomalia.7 := 0; 
END_IF;

//-------------------------------------------------------------------------------------------//
//----------------------------Anomalia rompimiento encoder de hilo---------------------------//
//-------------------------------------------------------------------------------------------//
IF (Encoder > (gEncoder_AbsolutoExtendido + 2000)) THEN
	gSupE_AnomaliasEntrada[32] := 0;
ELSE
	gSupE_AnomaliasEntrada[32] := 1;
END_IF

//-------------------------------------------------------------------------------------------//
//-------------------------------------Anchura E-Frame---------------------------------------//
//-------------------------------------------------------------------------------------------//
AnchoEFrame := 1600;

//-------------------------------------------------------------------------------------------//
//------Identificacion del estado inicial del E-Frame cuando tenemos una orden del AGV-------//
//-------------------------------------------------------------------------------------------//
IF I_OrdenCarga AND (NOT I_OrdenDescarga) AND (NOT I_OrdenDescargaB) AND (AUX_CONT_Automatico <>1) THEN
	OPT := init_descargado;
	Laser := Bumper;
	Opt_Carga := 1;
	Opt_Carga_ANT := 0;
	AUX_CONT_Automatico := 1;

ELSIF I_OrdenDescarga AND(NOT I_OrdenCarga) AND (NOT I_OrdenDescargaB) AND (AUX_CONT_Automatico <>1) THEN
	OPT := init_cargado;
	Laser := Bumper;
	Opt_Descarga := 1;
	Opt_Descarga_ANT:=0;
	AUX_CONT_Automatico := 1;
	
ELSIF I_OrdenDescargaB AND I_OrdenDescarga AND (NOT I_OrdenCarga) AND (AUX_CONT_Automatico <>1) THEN
	OPT := init_cargado_B;
	Laser := Bumper;
	Opt_Descarga_B := 1;
	Opt_DescargaB_ANT := 0;
	AUX_CONT_Automatico := 1;
END_IF

//-------------------------------------------------------------------------------------------//
//------------------------------Anomalia inductivos de la carga------------------------------//
//-------------------------------------------------------------------------------------------//
IF (gEstadoEframe = Automatico) AND (OPT = init_cargado) AND (Opt_Descarga < 5) AND ( ((NOT gEntradasPLC.DeteccionCarga1) AND (NOT gEntradasPLC.DeteccionCarga2)) 
 OR ((NOT gEntradasPLC.DeteccionCarga1) AND gEntradasPLC.DeteccionCarga2) OR (gEntradasPLC.DeteccionCarga1 AND (NOT gEntradasPLC.DeteccionCarga2)) ) THEN
	PalabraAnomalia.4 := 0;
ELSIF (gEstadoEframe = Automatico) AND (OPT = init_descargado) AND (Opt_Carga > 6) AND ( ((NOT gEntradasPLC.DeteccionCarga1) AND (NOT gEntradasPLC.DeteccionCarga2)) 
 OR ((NOT gEntradasPLC.DeteccionCarga1) AND gEntradasPLC.DeteccionCarga2) OR (gEntradasPLC.DeteccionCarga1 AND (NOT gEntradasPLC.DeteccionCarga2)) ) THEN
	PalabraAnomalia.4 := 0;
ELSIF (gEstadoEframe = Automatico) AND (OPT = init_cargado_B) AND (Opt_Descarga_B < 5) AND ( ((NOT gEntradasPLC.DeteccionCarga1) AND (NOT gEntradasPLC.DeteccionCarga2)) 
 OR ((NOT gEntradasPLC.DeteccionCarga1) AND gEntradasPLC.DeteccionCarga2) OR (gEntradasPLC.DeteccionCarga1 AND (NOT gEntradasPLC.DeteccionCarga2)) ) THEN
	PalabraAnomalia.4 := 0;
ELSE
	PalabraAnomalia.4 := 1;	
END_IF

IF (gEstadoEframe = Automatico) AND (OPT = init_cargado) AND (Opt_Descarga > 6) AND( (gEntradasPLC.DeteccionCarga1 AND gEntradasPLC.DeteccionCarga2) 
  OR ((NOT gEntradasPLC.DeteccionCarga1) AND gEntradasPLC.DeteccionCarga2) OR (gEntradasPLC.DeteccionCarga1 AND (NOT gEntradasPLC.DeteccionCarga2)) ) THEN
	PalabraAnomalia.1 := 0;	
ELSIF (gEstadoEframe = Automatico) AND (OPT = init_descargado) AND (Opt_Carga < 4) AND( (gEntradasPLC.DeteccionCarga1 AND gEntradasPLC.DeteccionCarga2) 
  OR ((NOT gEntradasPLC.DeteccionCarga1) AND gEntradasPLC.DeteccionCarga2) OR (gEntradasPLC.DeteccionCarga1 AND (NOT gEntradasPLC.DeteccionCarga2)) ) THEN
  	PalabraAnomalia.1 := 0;	
ELSIF (gEstadoEframe = Automatico) AND (OPT = init_cargado_B) AND (Opt_Descarga_B > 6) AND( (gEntradasPLC.DeteccionCarga1 AND gEntradasPLC.DeteccionCarga2) 
  OR ((NOT gEntradasPLC.DeteccionCarga1) AND gEntradasPLC.DeteccionCarga2) OR (gEntradasPLC.DeteccionCarga1 AND (NOT gEntradasPLC.DeteccionCarga2)) ) THEN
  	PalabraAnomalia.1 := 0;	
ELSE
	PalabraAnomalia.1 := 1;	
END_IF

//-------------------------------------------------------------------------------------------//
//--------------------------------------Control Automatico-----------------------------------//
//-------------------------------------------------------------------------------------------//
CASE OPT OF
	init_cargado:
		CASE Opt_Descarga OF
			1: // Comproba que el E-Frame esté en modo automatico y que tiene orden de descarga
				IF (gEntradasPLC.ModoAutomatico OR (gEstadoEframe = Reposo)) AND I_OrdenDescarga AND gEntradasPLC.Laser_OSSD1 AND gEntradasPLC.Laser_OSSD2 AND (AnchoEFrame = 1600) THEN
					Laser := Ext_con_carga_1600;
					Opt_Descarga_ANT := 1;
					Opt_Descarga := 2;
				ELSIF (gEntradasPLC.ModoAutomatico OR (gEstadoEframe = Reposo)) AND I_OrdenDescarga AND gEntradasPLC.Laser_OSSD1 AND gEntradasPLC.Laser_OSSD2 AND (AnchoEFrame = 1800) THEN
					Laser := Ext_con_carga_1800;
					Opt_Descarga_ANT := 1;
					Opt_Descarga := 2;
				END_IF
				
			2:  // Comproba que tiene condiciones para empezar el movimiento de extension del brazo
				IF (Opt_Descarga = 2) AND (Opt_Descarga_ANT = 1) THEN
					IF gEntradasPlc.InductivoBrazoRec AND (NOT gEntradasPlc.InductivoBrazoExt) AND (NOT gEntradasPLC.ParadaPrecisaBrazo) AND gEntradasPLC.InductivoSubirLevas
					 AND (NOT gEntradasPLC.InductivoBajarLevas) AND gEntradasPLC.DeteccionCarga1 AND gEntradasPLC.DeteccionCarga2 THEN
						AccionBrazo := A_Extender;
						gVelocidad := E_Cargado_Tramo1;
						
					//-----Anomalia inductivos de carga-----//
					ELSIF ((NOT gEntradasPLC.DeteccionCarga1) AND gEntradasPLC.DeteccionCarga2) OR (gEntradasPLC.DeteccionCarga1 AND (NOT gEntradasPLC.DeteccionCarga2)) OR
					 ((NOT gEntradasPLC.DeteccionCarga1) AND (NOT gEntradasPLC.DeteccionCarga2)) THEN
						PalabraAnomalia.4 := 0;	
					END_IF
					
					IF (Encoder < E_Tramo1) AND (Encoder > E_Tramo2) AND (AccionBrazo = A_Extender) THEN
						gVelocidad := E_Cargado_Tramo2;
						Opt_Descarga := 3;
						Opt_Descarga_ANT := 2;
					END_IF
				END_IF
				
			3:  // Controlo de la velocidad del E-Frame de acuerdo con su posicion
				IF (Opt_Descarga = 3) AND (Opt_Descarga_ANT = 2) THEN
					IF (Encoder < E_Tramo2) AND (AccionBrazo = A_Extender)  THEN
						gVelocidad := E_Cargado_Tramo3;
						Opt_Descarga := 4;
						Opt_Descarga_ANT := 3;
					END_IF
				END_IF	
			
			4:  // Verificacion de la deteccion de la fotocelula
				IF (Opt_Descarga = 4) AND (Opt_Descarga_ANT = 3) THEN
					IF (gEntradasPLC.ParadaPrecisaBrazo OR gEntradasPlc.InductivoBrazoExt) AND (AccionBrazo = A_Extender)  THEN
						Opt_Descarga := 5;
						Opt_Descarga_ANT := 4;
					END_IF
				END_IF
				
			5:  // Parada del motor y levas bajas
				IF (Opt_Descarga = 5) AND (Opt_Descarga_ANT = 4) THEN
					IF (NOT gEntradasPLC.ParadaPrecisaBrazo) AND gEntradasPlc.InductivoBrazoExt AND (AccionBrazo = A_Extender) THEN	
						AccionBrazo := A_Parar;
						gSupE_AnomaliasEntrada[33] := 0;
						
					ELSIF (gEntradasPLC.ParadaPrecisaBrazo AND gEntradasPLC.InductivoSubirLevas AND (NOT gEntradasPLC.InductivoBajarLevas) AND (NOT AUX_InitBajarLevas) ) AND (NOT AUX_EFrameDescargado) 
					  AND (AccionBrazo = A_Extender) THEN   
						IF ((NOT gEntradasPLC.DeteccionCarga1) AND (NOT gEntradasPLC.DeteccionCarga2)) OR ((NOT gEntradasPLC.DeteccionCarga1) AND gEntradasPLC.DeteccionCarga2) OR
						(gEntradasPLC.DeteccionCarga1 AND (NOT gEntradasPLC.DeteccionCarga2)) THEN
							PalabraAnomalia.4 := 0;	
						ELSIF gEntradasPLC.DeteccionCarga1 AND gEntradasPLC.DeteccionCarga2 THEN
							AccionBrazo := A_Parar;
							gEstadoLevas := bajar;
							AUX_EFrameDescargado := TRUE; 
						END_IF
					END_IF
					
					IF (NOT gEntradasPlc.InductivoBrazoExt) THEN
						ACC03_ControlLevas();
					END_IF

					//----- Anomalia cuando no detecta inductivo y si encuentra en un rango de encoder de hilo -----//
					IF (NOT gEntradasPlc.InductivoBrazoExt) AND (Encoder < (Encoder_Extendido + Encoder_Extendido_OFFSET) ) AND (Encoder > (Encoder_Extendido - Encoder_Extendido_OFFSET)) THEN
						AccionBrazo := A_Parar;
						PalabraAnomalia.5 := 0;	
					END_IF
					
					IF LevasAbajoDONE AND gEntradasPLC.ParadaPrecisaBrazo AND (NOT gEntradasPLC.InductivoSubirLevas) AND gEntradasPLC.InductivoBajarLevas THEN
						LevasAbajoDONE := FALSE;
						AUX_EFrameDescargado := FALSE;
						Opt_Descarga := 6;
						Opt_Descarga_ANT := 5;
					END_IF
				END_IF
				
			6:  // Recoja del brazo despues de la descarga 
				IF (Opt_Descarga = 6) AND (Opt_Descarga_ANT = 5) THEN
					AccionBrazo := A_Recoger;
					gVelocidad := R_Descargado_Tramo2;
					Laser := Bumper;

					IF (Encoder > E_Tramo1) AND (AccionBrazo = A_Recoger) THEN
						gVelocidad := R_Descargado_Tramo1;
						Opt_Descarga := 7;
						Opt_Descarga_ANT := 6;
					END_IF
				END_IF
				
			7:  // Reduzir la velocidad del brazo
				IF (Opt_Descarga = 7) AND (Opt_Descarga_ANT = 6) THEN
					IF gEntradasPlc.InductivoBrazoRec AND (AccionBrazo = A_Recoger) THEN  
						Opt_Descarga := 8;
						Opt_Descarga_ANT := 7;
						I_OrdenDescarga := FALSE;
						
					//----- Anomalia para el caso de no detectar inductivos y encoder de hilo en un determinado rango -----//
					ELSIF (NOT gEntradasPlc.InductivoBrazoRec) AND (Encoder > (gEncoder_Absoluto - Encoder_Recogido_OFFSET)) AND (Encoder < (gEncoder_Absoluto + Encoder_Recogido_OFFSET)) AND (AccionBrazo = A_Recoger) THEN
						AccionBrazo := A_Parar;
						PalabraAnomalia.6 := 0;
					END_IF
				END_IF
				
			8:  // Fin de la operativa de descarga
				IF (Opt_Descarga = 8) AND (Opt_Descarga_ANT = 7) THEN
					gVelocidad := SinConsigna;
					AccionBrazo := A_Parar;
					gEstadoEframe := Reposo;
					I_OrdenDescarga := FALSE;
					gCargaOPT := 2;
					ESTADOS();
					Init_EstadoCarga := FALSE;
					AUX_CONT_Automatico := 0;
					Opt_Descarga := 1;
					Opt_Descarga_ANT:=0;
					Laser := Bumper;
					OPT := indeterminado_OPT;
				END_IF
		END_CASE
		
	init_descargado:
		CASE Opt_Carga OF
			1:  // Comproba que el E-Frame esté en modo automatico y que tiene orden de carga
				IF (gEntradasPLC.ModoAutomatico OR (gEstadoEframe = Reposo)) AND I_OrdenCarga AND gEntradasPLC.Laser_OSSD1 AND gEntradasPLC.Laser_OSSD2 THEN
					Laser := Ext_sin_carga;
					Opt_Carga_ANT := 1;
					Opt_Carga := 2;
				END_IF

			2:  // Comproba que tiene condiciones para empezar el movimiento de extension del brazo
				IF (Opt_Carga = 2) AND (Opt_Carga_ANT = 1)  THEN 
					IF gEntradasPlc.InductivoBrazoRec AND (NOT gEntradasPlc.InductivoBrazoExt) AND (NOT gEntradasPLC.ParadaPrecisaBrazo) AND (NOT gEntradasPLC.InductivoSubirLevas)
					 AND gEntradasPLC.InductivoBajarLevas AND (NOT gEntradasPLC.DeteccionCarga1) AND (NOT gEntradasPLC.DeteccionCarga2) THEN 
						AccionBrazo := A_Extender;
						gVelocidad := E_Descargado_Tramo1;
						
					//----- Anomalia inductivos de carga -----//
					ELSIF ((NOT gEntradasPLC.DeteccionCarga1) AND gEntradasPLC.DeteccionCarga2) OR (gEntradasPLC.DeteccionCarga1 AND (NOT gEntradasPLC.DeteccionCarga2)) OR
					 (gEntradasPLC.DeteccionCarga1 AND gEntradasPLC.DeteccionCarga2) THEN
						PalabraAnomalia.4 := 0;		
					END_IF
	
					IF (Encoder < E_Tramo1) AND (Encoder > E_Tramo2) AND (AccionBrazo = A_Extender) THEN
						gVelocidad := E_Descargado_Tramo2;
						Opt_Carga := 3;
						Opt_Carga_ANT := 2;
					END_IF
				END_IF

			3:  // Controlo de la velocidad del E-Frame de acuerdo con su posicion
				IF (Opt_Carga = 3) AND (Opt_Carga_ANT = 2)  THEN
					IF ((Encoder < E_Tramo2) OR gEntradasPLC.DeteccionCargaExt) AND (AccionBrazo = A_Extender) THEN
						gVelocidad := E_Descargado_Tramo3;
						Opt_Carga := 4;
						Opt_Carga_ANT := 3;
					END_IF
				END_IF	

			4:  // Verificacion de la deteccion de la fotocelula
				IF (Opt_Carga = 4) AND (Opt_Carga_ANT = 3) THEN
					IF gEntradasPLC.DeteccionCarga1 AND gEntradasPLC.DeteccionCarga2 THEN
						IF (NOT ParadaLaser) THEN
							AUX_DetecionCarga := TRUE;
							TON_DetecionCarga( IN:=AUX_DetecionCarga, PT:=T#500MS, ET => Tempo_Actual_DetecionCarga);
						ELSIF ParadaLaser THEN
							AUX_DetecionCarga := TRUE;
							TON_DetecionCarga( IN:=AUX_DetecionCarga, PT:=T#1S, ET => Tempo_Actual_DetecionCarga);
						END_IF
						
						IF TON_DetecionCarga.Q AND (NOT gEntradasPLC.ParadaPrecisaBrazo) AND AUX_DetecionCarga THEN
							gSupE_AnomaliasEntrada[35] := 0;
							
						ELSIF (NOT TON_DetecionCarga.Q) AND (gEntradasPLC.ParadaPrecisaBrazo OR gEntradasPlc.InductivoBrazoExt) AND (AccionBrazo = A_Extender) THEN
							Opt_Carga := 5;
							Opt_Carga_ANT := 4;
						END_IF
					ELSIF ( ((NOT gEntradasPLC.DeteccionCarga1) AND (NOT gEntradasPLC.DeteccionCarga2)) OR ((NOT gEntradasPLC.DeteccionCarga1) AND gEntradasPLC.DeteccionCarga2) OR
						(gEntradasPLC.DeteccionCarga1 AND (NOT gEntradasPLC.DeteccionCarga2)) ) AND (gEntradasPLC.ParadaPrecisaBrazo OR gEntradasPlc.InductivoBrazoExt) AND (AccionBrazo = A_Extender) THEN
						Opt_Carga := 5;	
						Opt_Carga_ANT := 4;
					END_IF 
				END_IF

			5:  // Subir Levas despues de parar el brazo en la fotocelula
				IF (Opt_Carga = 5) AND (Opt_Carga_ANT = 4) THEN
					IF (NOT gEntradasPLC.ParadaPrecisaBrazo) AND gEntradasPlc.InductivoBrazoExt AND (AccionBrazo = A_Extender) THEN	
						gSupE_AnomaliasEntrada[33] := 0;
						
					ELSIF (gEntradasPLC.ParadaPrecisaBrazo AND (NOT gEntradasPLC.InductivoSubirLevas) AND gEntradasPLC.InductivoBajarLevas AND (NOT AUX_InitSubirLevas)) AND (AccionBrazo = A_Extender) THEN
						AUX_DetecionCarga := FALSE;
						TON_DetecionCarga(IN:=FALSE);
						
						IF ((NOT gEntradasPLC.DeteccionCarga1) AND (NOT gEntradasPLC.DeteccionCarga2)) OR ((NOT gEntradasPLC.DeteccionCarga1) AND gEntradasPLC.DeteccionCarga2) OR
						(gEntradasPLC.DeteccionCarga1 AND (NOT gEntradasPLC.DeteccionCarga2)) THEN
							PalabraAnomalia.4 := 0;	
						ELSIF gEntradasPLC.DeteccionCarga1 AND gEntradasPLC.DeteccionCarga2 THEN
							ParadaFotocelula := TRUE;
							AccionBrazo := A_Parar;
							gEstadoLevas := subir;
							AUX_InitSubirLevas := TRUE; 
						END_IF 
					END_IF
					
					IF (NOT gEntradasPlc.InductivoBrazoExt) THEN
						ACC03_ControlLevas();
					END_IF

					//----- Anomalia para el caso de no detectar inductivos y encoder de hilo en un determinado rango -----//
					IF (NOT gEntradasPlc.InductivoBrazoExt) AND (Encoder < (Encoder_Extendido + Encoder_Extendido_OFFSET) ) AND (Encoder > (Encoder_Extendido - Encoder_Extendido_OFFSET)) THEN
						AccionBrazo := A_Parar;
						PalabraAnomalia.5 := 0;
					END_IF
	
					IF LevasArribaDONE AND gEntradasPLC.ParadaPrecisaBrazo AND gEntradasPLC.InductivoSubirLevas AND (NOT gEntradasPLC.InductivoBajarLevas) THEN
						LevasArribaDONE := FALSE;
						Opt_Carga := 6;
						Opt_Carga_ANT := 5;
					END_IF
				END_IF
				
			6:  // Recoja del brazo despues de la carga
				IF (Opt_Carga = 6) AND (Opt_Carga_ANT = 5) THEN
					AUX_InitSubirLevas := FALSE;
					AccionBrazo := A_Recoger;
					gVelocidad := R_Cargado_Tramo3;
					Laser := Bumper;

					IF (Encoder > E_Tramo2) AND (Encoder < E_Tramo1) AND (AccionBrazo = A_Recoger) THEN
						gVelocidad := R_Cargado_Tramo2;
						Opt_Carga := 7;
						Opt_Carga_ANT := 6;
					END_IF
				END_IF

			7:  // Cambio de la velocidad del brazo
				IF (Opt_Carga = 7) AND (Opt_Carga_ANT = 6) THEN
					IF (Encoder > E_Tramo1) AND (AccionBrazo = A_Recoger) THEN
						gVelocidad := R_Cargado_Tramo1;
						Opt_Carga := 8;
						Opt_Carga_ANT := 7;
					END_IF
				END_IF

			8:  // Reduzir la velocidad del brazo
				IF (Opt_Carga = 8) AND (Opt_Carga_ANT = 7) THEN
					IF gEntradasPlc.InductivoBrazoRec AND (AccionBrazo = A_Recoger) THEN
						Opt_Carga := 9;
						Opt_Carga_ANT := 8;
						I_OrdenCarga := FALSE;
					ELSIF (NOT gEntradasPlc.InductivoBrazoRec) AND (Encoder > (gEncoder_Absoluto - Encoder_Recogido_OFFSET)) AND (Encoder < (gEncoder_Absoluto + Encoder_Recogido_OFFSET)) AND (AccionBrazo = A_Recoger) THEN
						AccionBrazo := A_Parar;
						PalabraAnomalia.6 := 0;
					END_IF
				END_IF

			9:  // Fin de la operativa de descarga
				IF (Opt_Carga = 9) AND (Opt_Carga_ANT = 8) THEN
					AUX_InitSubirLevas := FALSE;
					gVelocidad := SinConsigna;
					AccionBrazo := A_Parar;
					gEstadoEframe := Reposo; 
					I_OrdenCarga := FALSE;
					gCargaOPT := 1;	
					ESTADOS();
					AUX_CONT_Automatico := 0;
					Opt_Carga := 1;	
					Opt_Carga_ANT := 0;
					Laser := Bumper;
					OPT := indeterminado_OPT;
					ParadaLaser := FALSE;
				END_IF
		END_CASE
		
	init_cargado_B:
		CASE Opt_Descarga_B OF
			1:  // Comproba que el E-Frame esté en modo automatico y que tiene orden de descarga
				IF (gEntradasPLC.ModoAutomatico OR (gEstadoEframe = Reposo)) AND I_OrdenDescargaB AND gEntradasPLC.Laser_OSSD1 AND gEntradasPLC.Laser_OSSD2 AND (AnchoEFrame = 1600) THEN
					Laser := Ext_con_carga_1600;
					Opt_DescargaB_ANT := 1;
					Opt_Descarga_B := 2;
				ELSIF (gEntradasPLC.ModoAutomatico OR (gEstadoEframe = Reposo)) AND I_OrdenDescargaB AND gEntradasPLC.Laser_OSSD1 AND gEntradasPLC.Laser_OSSD2 AND (AnchoEFrame = 1800) THEN
					Laser := Ext_con_carga_1800;
					Opt_DescargaB_ANT := 1;
					Opt_Descarga_B := 2;
				END_IF

			2:  // Comproba que tiene condiciones para empezar el movimiento de extension del brazo
				IF (Opt_Descarga_B = 2) AND (Opt_DescargaB_ANT = 1)  THEN 
					IF gEntradasPlc.InductivoBrazoRec AND (NOT gEntradasPlc.InductivoBrazoExt) AND (NOT gEntradasPLC.ParadaPrecisaBrazo) AND gEntradasPLC.InductivoSubirLevas
					 AND (NOT gEntradasPLC.InductivoBajarLevas) AND gEntradasPLC.DeteccionCarga1 AND gEntradasPLC.DeteccionCarga2 THEN 
						AccionBrazo := A_Extender;
						gVelocidad := E_Cargado_Tramo1;
						
					//----- Anomalia inductivos de carga -----//
					ELSIF ((NOT gEntradasPLC.DeteccionCarga1) AND gEntradasPLC.DeteccionCarga2) OR (gEntradasPLC.DeteccionCarga1 AND (NOT gEntradasPLC.DeteccionCarga2)) OR
					 ((NOT gEntradasPLC.DeteccionCarga1) AND (NOT gEntradasPLC.DeteccionCarga2)) THEN
						PalabraAnomalia.4 := 0;	
					END_IF
					
					IF (Encoder < E_Tramo1) AND (Encoder > E_Tramo2) AND (AccionBrazo = A_Extender) THEN
						gVelocidad := E_Cargado_Tramo2;
						Opt_Descarga_B := 3;
						Opt_DescargaB_ANT := 2;
					END_IF
				END_IF

			3:  // Controlo de la velocidad del E-Frame de acuerdo con su posicion
				IF (Opt_Descarga_B = 3) AND (Opt_DescargaB_ANT = 2) THEN
					IF (Encoder < E_Tramo2) AND (AccionBrazo = A_Extender)  THEN
						gVelocidad := E_Cargado_Tramo3;
						Opt_Descarga_B := 4;
						Opt_DescargaB_ANT := 3;
					END_IF
				END_IF	

			4:   // Verificacion del valor del encoder
				IF (Opt_Descarga_B = 4) AND (Opt_DescargaB_ANT = 3) THEN
					OPT_Retener := 1;
					
					IF ((Encoder < (Encoder_Parada + Encoder_Parada_OFFSET)) AND (Encoder > (Encoder_Parada - Encoder_Parada_OFFSET)) OR gEntradasPlc.InductivoBrazoExt) AND (AccionBrazo = A_Extender)  THEN
						Opt_Descarga_B := 5;
						Opt_DescargaB_ANT := 4;
					END_IF
				END_IF

			5:  // Parada del motor y levas bajas
				IF (Opt_Descarga_B = 5) AND (Opt_DescargaB_ANT = 4) THEN
					IF gEntradasPlc.InductivoBrazoExt AND (AccionBrazo = A_Extender) THEN	
						AccionBrazo := A_Parar;
						gSupE_AnomaliasEntrada[33] := 0;
						
					ELSIF (Encoder < (Encoder_Parada + Encoder_Parada_OFFSET)) AND (Encoder > (Encoder_Parada - Encoder_Parada_OFFSET)) AND (NOT AUX_InitBajarLevas) AND (NOT AUX_EFrameDescargado) 
					  AND (AccionBrazo = A_Extender) AND gEntradasPLC.InductivoSubirLevas AND (NOT gEntradasPLC.InductivoBajarLevas) THEN 
						IF ((NOT gEntradasPLC.DeteccionCarga1) AND (NOT gEntradasPLC.DeteccionCarga2)) OR ((NOT gEntradasPLC.DeteccionCarga1) AND gEntradasPLC.DeteccionCarga2) OR
						  (gEntradasPLC.DeteccionCarga1 AND (NOT gEntradasPLC.DeteccionCarga2)) THEN
							PalabraAnomalia.4 := 0;	
						ELSIF gEntradasPLC.DeteccionCarga1 AND gEntradasPLC.DeteccionCarga2 THEN
							AccionBrazo := A_Parar;
							gEstadoLevas := bajar;
							AUX_EFrameDescargado := TRUE; 
						END_IF
					END_IF
					
					IF (NOT gEntradasPlc.InductivoBrazoExt) THEN
						ACC03_ControlLevas();
					END_IF

					//----- Anomalia cuando no detecta inductivo y si encuentra en un rango de encoder de hilo -----/
					IF (NOT gEntradasPlc.InductivoBrazoExt) AND (Encoder < (Encoder_Extendido + Encoder_Extendido_OFFSET) ) AND (Encoder > (Encoder_Extendido - Encoder_Extendido_OFFSET)) THEN
						AccionBrazo := A_Parar;
						PalabraAnomalia.5 := 0;	
					END_IF
					
					IF LevasAbajoDONE AND (NOT gEntradasPLC.InductivoSubirLevas) AND gEntradasPLC.InductivoBajarLevas THEN
						LevasAbajoDONE := FALSE;
						AUX_EFrameDescargado := FALSE;
						Opt_Descarga_B := 6;
						Opt_DescargaB_ANT := 5;
					END_IF
				END_IF

			6:  // Recoja del brazo despues de la descarga
				IF (Opt_Descarga_B = 6) AND (Opt_DescargaB_ANT = 5) THEN
					AccionBrazo := A_Recoger;
					gVelocidad := R_Descargado_Tramo2;
					Laser := Bumper;
					
					IF (Encoder > E_Tramo1) AND (AccionBrazo = A_Recoger) THEN
						gVelocidad := R_Descargado_Tramo1;
						Opt_Descarga_B := 7;
						Opt_DescargaB_ANT := 6;
					END_IF
				END_IF

			7:  // Reduzir la velocidad del brazo
				IF (Opt_Descarga_B = 7) AND (Opt_DescargaB_ANT = 6) THEN
					IF gEntradasPlc.InductivoBrazoRec AND (AccionBrazo = A_Recoger) THEN  
						Opt_Descarga_B := 8;
						Opt_DescargaB_ANT := 7;
						I_OrdenDescargaB := FALSE;
						I_OrdenDescarga := FALSE;
						
					//----- Anomalia para el caso de no detectar inductivos y encoder de hilo en un determinado rango -----//
					ELSIF (NOT gEntradasPlc.InductivoBrazoRec) AND (Encoder > (gEncoder_Absoluto - Encoder_Recogido_OFFSET)) AND (Encoder < (gEncoder_Absoluto + Encoder_Recogido_OFFSET)) AND (AccionBrazo = A_Recoger) THEN
						AccionBrazo := A_Parar;
						PalabraAnomalia.6 := 0;
					END_IF
				END_IF

			8:  // Fin de la operativa de descarga
				IF (Opt_Descarga_B = 8) AND (Opt_DescargaB_ANT = 7) THEN
					AccionBrazo := A_Parar;
					gVelocidad := SinConsigna;
					gEstadoEframe := Reposo;
					I_OrdenDescargaB := FALSE;
					I_OrdenDescarga := FALSE;
					gCargaOPT := 2;
					ESTADOS();
					Init_EstadoCarga := FALSE;
					AUX_CONT_Automatico := 0;
					Opt_Descarga_B := 1;
					Opt_DescargaB_ANT := 0;
					Laser := Bumper;
					OPT := indeterminado_OPT;
				END_IF
		END_CASE
END_CASE	

//-------------------------------------------------------------------------------------------//
//------------------------------Asignacion de anomalias del supervisor-----------------------//
//-------------------------------------------------------------------------------------------//
gSupE_AnomaliasEntrada[18] := PalabraAnomalia.0;
gSupE_AnomaliasEntrada[19] := PalabraAnomalia.1;
gSupE_AnomaliasEntrada[20] := PalabraAnomalia.2;
gSupE_AnomaliasEntrada[22] := PalabraAnomalia.4;
gSupE_AnomaliasEntrada[23] := PalabraAnomalia.5;
gSupE_AnomaliasEntrada[24] := PalabraAnomalia.6;
gSupE_AnomaliasEntrada[25] := PalabraAnomalia.7;

END_PROGRAM

// StandardPLC/Application/CÓDIGO/Sub ACCIONES/ACC03_ControlLevas
PROGRAM ACC03_ControlLevas
VAR
	// Variables para control de los tiempos para subir y bajar levas
	Tempo_Actual_BajarLevas 		:TIME;
	Tempo_Actual 					:TIME;
	
	// Variable para inicializar solo una vez el timer
	Init_Timer						:BOOL;
END_VAR

(*//////////////////////////////////////////////////////////////////////////////////////////////////////////////////////////////////////////////////////////////////////////////////////////////////////////////////////////////////////////////////
ACC03_ControlLevas (PRG)                      

Description:	Control de las levas en modo automatico
				Existen 3 estados para las levas: subir, bajar y apagado
		 
///////////////////////////////////////////////////////////////////////////////////////////////////////////////////////////////////////////////////////////////////////////////////////////////////////////////////////////////////////////////////// *)

//-------------------------------------------------------------------------------------------//
//------------------------------Anomalia de los inductivos de carga--------------------------//
//-------------------------------------------------------------------------------------------//
IF ((NOT gEntradasPLC.DeteccionCarga1) AND (NOT gEntradasPLC.DeteccionCarga2)) OR ((NOT gEntradasPLC.DeteccionCarga1) AND gEntradasPLC.DeteccionCarga2) OR
	(gEntradasPLC.DeteccionCarga1 AND (NOT gEntradasPLC.DeteccionCarga2)) AND (gEstadoLevas = subir) THEN
		PalabraAnomalia.4 := 0;	
END_IF

//-------------------------------------------------------------------------------------------//
//-------------------------------------Control de las levas----------------------------------//
//-------------------------------------------------------------------------------------------//
CASE gEstadoLevas OF
	subir:
		CASE control_subir OF
			1:  // Inicia el movimiento de subida de las levas
				IF ParadaFotocelula AND gEntradasPLC.DeteccionCarga1 AND gEntradasPLC.DeteccionCarga2 THEN
					gSalidasPLC.SubirLevas := TRUE;
					control_subir := 2;
				END_IF
				
			2:  // Para el movimiento de subida de las levas
				AUX_SubirLevas := TRUE;
				TON_SubirLevas(IN:=AUX_SubirLevas, PT:=T#4S, ET => Tempo_Actual);
				
				IF TON_SubirLevas.Q THEN
					gSalidasPLC.SubirLevas := FALSE;

					//----- Anomalia en las levas -----//
					IF ((NOT gEntradasPLC.InductivoSubirLevas) AND (NOT gEntradasPLC.InductivoBajarLevas)) OR
				      (gEntradasPLC.InductivoSubirLevas AND gEntradasPLC.InductivoBajarLevas) THEN
						gSupE_AnomaliasEntrada[21] := 0;
						gEstadoLevas := apagado;
					ELSE
						AUX_SubirLevas := FALSE;
						TON_SubirLevas(IN:=FALSE);
						control_subir := control_subir := 3;
					END_IF	
				END_IF

			3:  // Analisa si tenemos anomalia en las levas
				LevasArribaDONE:=TRUE;
				ParadaFotocelula := FALSE;
				
				//----- Anomalia en las levas -----//
				IF ((NOT gEntradasPLC.InductivoSubirLevas) AND (NOT gEntradasPLC.InductivoBajarLevas)) OR
				  (gEntradasPLC.InductivoSubirLevas AND gEntradasPLC.InductivoBajarLevas) THEN
					gSupE_AnomaliasEntrada[21] := 0;
					gEstadoLevas := apagado;
				ELSE
					control_subir := 1;
					gEstadoLevas := apagado;
				END_IF
		END_CASE
	
	bajar:
		CASE control_bajar OF
			1:  // Inicia el motor para bajar levas
				IF gEntradasPLC.InductivoSubirLevas AND (NOT gEntradasPLC.InductivoBajarLevas) AND (NOT AUX_InitBajarLevas)  THEN
					gSalidasPLC.BajarLevas := TRUE;
					AUX_InitBajarLevas := TRUE;
					control_bajar := 2;
				END_IF
				
			2:  // Inicia el timer de bajar levas. Cuanto timer completo, cambia de estado
				AUX_BajarLevas := TRUE;
				TON_BajarLevas( IN:=AUX_BajarLevas, PT:=T#4S, ET => Tempo_Actual_BajarLevas);
				
				IF TON_BajarLevas.Q THEN
					gSalidasPLC.BajarLevas := FALSE;
					
					//----- Anomalia en las levas -----//
					IF ((NOT gEntradasPLC.InductivoSubirLevas) AND (NOT gEntradasPLC.InductivoBajarLevas)) OR (gEntradasPLC.InductivoSubirLevas AND (NOT gEntradasPLC.InductivoBajarLevas)) THEN
						gSupE_AnomaliasEntrada[21] := 0;
						gEstadoLevas := apagado;
					ELSE
						AUX_BajarLevas := FALSE;
						TON_BajarLevas(IN:=FALSE);
						control_bajar := 3;
					END_IF	
				END_IF

			3:  // Desliga el motor y resetea las variables
				AUX_InitBajarLevas := FALSE;
				LevasAbajoDONE := TRUE;
				
				//----- Anomalia en las levas -----//
				IF ((NOT gEntradasPLC.InductivoSubirLevas) AND (NOT gEntradasPLC.InductivoBajarLevas)) OR (gEntradasPLC.InductivoSubirLevas AND (NOT gEntradasPLC.InductivoBajarLevas)) THEN
					gSupE_AnomaliasEntrada[21] := 0;
					gEstadoLevas := apagado;
				ELSE
					control_bajar := 1;
					gEstadoLevas := apagado;
				END_IF
		END_CASE

	apagado:  // Motor de las levas apagado
		gSalidasPLC.SubirLevas := FALSE;
		gSalidasPLC.BajarLevas := FALSE;
		AUX_SubirLevas := FALSE;
		TON_SubirLevas(IN:=FALSE);
		AUX_BajarLevas := FALSE;
		TON_BajarLevas(IN:=FALSE);
END_CASE

END_PROGRAM

// StandardPLC/Application/CÓDIGO/Sub Dispositivos/DISP01_CntrlExtensionGeneral_FB
FUNCTION_BLOCK DISP01_CntrlExtensionGeneral_FB
VAR_INPUT
	I_TIEMPO_SEGURIDAD 		:TIME;	        //----- Tiempo máximo de un movimiento despliegue/contracción, incluyendo margen seguridad -----//	
	I_CLEAR			   		:BOOL;
	I_RESET			   		:BOOL;			//----- Reset módulo. En alta desactiva salidas, identifica estado y limpia anomalías. -----//	
	I_HABILITAR		   		:BOOL;			//----- Entrada para habilitar salidas control. Podemos usar como condición de seguridad. -----//	

	I_DetecExtend			:BOOL;
	I_DetectRecog			:BOOL;
END_VAR
VAR_OUTPUT
	O_Estado				:BYTE;
	O_Anomalia				:BYTE;
END_VAR
VAR
	EstadoAnomalia			:BYTE := 16#FF;
	EstadoExtension			:BYTE;

	TONDEV_0				:TON;
	TONDEV_1				:TON;
	TONDEV_2				:TON;
	TONDEV_3				:TON;
	TONDEV_E				:TON;
	TONDEV_R				:TON;
	
	//----- Variables para el control de los tiempos -----//	
	Tiempo_Ext				:TIME;
	Tiempo_Rec				:TIME;
END_VAR

(*//////////////////////////////////////////////////////////////////////////////////////////////////////////////////////////////////////////////////////////////////////////////////////////////////////////////////////////////////////////////////
DISP01_CntrlExtensionGeneral_FB (FB)                     

Description:	Control de anomalias en la extension o recoja del brazo.

				O_Estado := 0		-> Estado indeterminado
				O_Estado := 1		-> Brazo recogido
				O_Estado := 2		-> Brazo en estado intermedio
				O_Estado := 3		-> Brazo extendido

///////////////////////////////////////////////////////////////////////////////////////////////////////////////////////////////////////////////////////////////////////////////////////////////////////////////////////////////////////////////////// *)

IF I_RESET AND (NOT LASER_AUX) THEN
	EstadoAnomalia := 16#FF;
	EstadoExtension := 0;
	AccionBrazo := A_Parar;
END_IF;

IF I_CLEAR THEN 
	EstadoAnomalia := 16#FF; 
END_IF;

//----------------------Inabilita las acciones de extender y recoger del brazo---------------//
IF ( (EstadoAnomalia <> 16#FF) OR (NOT I_HABILITAR) ) AND (NOT LASER_AUX) THEN
	AccionBrazo := A_Parar;
END_IF;


//--------------------------Timers que van a ayudar a generar anomalias----------------------//
TONDEV_1( IN := ( (NOT (I_CLEAR OR I_RESET)) AND (I_DetecExtend OR (NOT I_DetectRecog)) AND (gEstadoEframe=Reposo)), PT := T#1S);    //----- El estado debería ser recogido pero se detecta en inductivo de extendido -----//	
TONDEV_2( IN := ( (NOT (I_CLEAR OR I_RESET)) AND (I_DetecExtend OR I_DetectRecog)), PT := T#1S);          //----- EL estado debería ser intermedio pero el brazo esta extendido o recogido -----//	
TONDEV_3( IN := ( (NOT (I_CLEAR OR I_RESET)) AND ((NOT I_DetecExtend) OR I_DetectRecog)), PT := T#1S);    //----- El brazo debería estar extendido pero esta recogido -----//	
	
CASE EstadoExtension OF
1:	// Estado Recogido
	IF ( ((AccionBrazo = A_Extender) OR (AccionBrazo = M_Extender) OR (AccionBrazo = Laser_Parar))  AND (NOT I_DetectRecog) ) THEN
		EstadoExtension := 2;
	ELSIF TONDEV_1.Q THEN
		EstadoExtension := 0;
		EstadoAnomalia.0 := 0;
	END_IF;
	
2:	// Estado Intermedio
	IF ( ((AccionBrazo = A_Extender) OR (AccionBrazo = M_Extender) OR (AccionBrazo = Laser_Parar) OR (AccionBrazo = A_Parar)) AND I_DetecExtend AND (NOT I_DetectRecog) ) THEN
		EstadoExtension := 3;
	ELSIF ( ((AccionBrazo = A_Recoger) OR (AccionBrazo = M_Parar)) AND (NOT I_DetecExtend) AND I_DetectRecog ) THEN
		EstadoExtension := 1;
	ELSIF TONDEV_2.Q THEN
		EstadoExtension := 0;
	END_IF;
	
3:	// Estado Extendido
	IF ( ((AccionBrazo = A_Recoger) OR (AccionBrazo = M_Recoger)) AND (NOT I_DetecExtend) ) THEN
		EstadoExtension := 2;
	ELSIF TONDEV_3.Q THEN
		EstadoExtension := 0;
		EstadoAnomalia.2 := 0;
	END_IF;
ELSE
	IF (EstadoAnomalia <> 16#FF) THEN
		EstadoExtension :=0;
	ELSIF I_DetecExtend AND NOT I_DetectRecog THEN
		EstadoExtension:=3;	
	ELSIF NOT I_DetecExtend AND NOT I_DetectRecog THEN
		EstadoExtension:=2;	
	ELSIF NOT I_DetecExtend AND I_DetectRecog THEN
		EstadoExtension:=1;	
	ELSE
		EstadoExtension := 0;
		EstadoAnomalia.3 := (I_CLEAR OR I_RESET);
	END_IF;
END_CASE

//----------------------------------Anomalía doble detección---------------------------------//
TONDEV_0( IN := ( (NOT (I_CLEAR OR I_RESET)) AND (I_DetecExtend AND I_DetectRecog)), PT := T#1S);
IF TONDEV_0.Q THEN 
	EstadoAnomalia.3 := 0; 
	EstadoExtension := 0; 
END_IF;

//-----------------------Anomalia por exceso de tiempo a extender/recoger--------------------//															
TONDEV_E(IN := ((AccionBrazo = A_Extender) OR (AccionBrazo = M_Extender)), PT := I_TIEMPO_SEGURIDAD, ET => Tiempo_Ext);
TONDEV_R(IN := ((AccionBrazo = A_Recoger) OR (AccionBrazo = M_Recoger)), PT := I_TIEMPO_SEGURIDAD, ET => Tiempo_Rec);
IF TONDEV_E.Q THEN 
	EstadoAnomalia.4 := 0; 
	EstadoExtension := 0; 
END_IF;
IF TONDEV_R.Q THEN 
	EstadoAnomalia.5 := 0; 
	EstadoExtension := 0; 
END_IF;
	
//-------------------------------------Salidas de la funcion---------------------------------//		
O_Anomalia := EstadoAnomalia;
O_Estado := EstadoExtension;

END_FUNCTION_BLOCK

// StandardPLC/Application/CÓDIGO/ACCIONES
PROGRAM ACCIONES
VAR
	TON_Extender				:TON;
	TON_Retraer					:TON;
	
	AUX_TIMER_Retraer			:BOOL;
	AUX_TIMER_Extender			:BOOL;
	ControlExtension			:DISP01_CntrlExtensionGeneral_FB;
END_VAR

(*/////////////////////////////////////////////////////////////////////////////////////////////////////////////////////////////////////////////////////////////////////////////////////////////////////////////////////////////////////////////////
ACCIONES (PRG)                     

Description:	Se llaman distintas funciones dependiendo del estado del E-Frame
				Es aquí donde controlamos el cambio de colores de la luz
 
///////////////////////////////////////////////////////////////////////////////////////////////////////////////////////////////////////////////////////////////////////////////////////////////////////////////////////////////////////////////////// *)

Setas_Seguridad();
Laser_Seguridad();

//-------------------------------------------------------------------------------------------//
//-----------------------Control de la baliza dependiendo del estado-------------------------//
//-------------------------------------------------------------------------------------------//
IF ( gFinEncendido ) THEN
	CASE gEstadoEframe OF
		Manual:
			ACC01_ControlManual();
			
			IF TeachingDone THEN
				Disp_SelectIndicadores := 15;			//----- Baliza verde y acustico constante -----//
			ELSE
				Disp_SelectIndicadores := 5;			//----- Baliza amarillo y rojo intermitente -----//	
			END_IF
			
		Degradado:
			ACC00_SalidasDesactivadas();
			Disp_SelectIndicadores := 5;				//----- Baliza amarillo y rojo intermitente -----//

		Reposo:
			Disp_SelectIndicadores := 2;				//----- Baliza verde -----//

		Automatico:
			IF (NOT LASER_AUX) THEN
				ACC02_ControlAutomatico( I_HABILITAR := gFinEncendido AND ((gEstadoEframe=Reposo) OR (gEstadoEframe=Automatico) OR (gEstadoEframe=Reinicio) OR (gEstadoEframe=Anomalia AND gSupS_ControlEstados=1) ),
						 I_OrdenCarga := gEntradasAGV.OrdenCarga AND (gEstadoEframe=Automatico),
						 I_OrdenDescarga := gEntradasAGV.OrdenDescarga AND (gEstadoEframe=Automatico),
						 I_OrdenDescargaB := gEntradasAGV.OrdenDescarga AND gEntradasAGV.OrdenDescargaB AND (gEstadoEframe=Automatico));
			
				Disp_SelectIndicadores := 3;			//----- Baliza amarillo -----//
			END_IF
			
		Anomalia:
			IF (gSupS_MensajeAnom = 1)  THEN
				Disp_SelectIndicadores := 13;
			ELSIF (gSupS_MensajeAnom = 2) THEN
				Disp_SelectIndicadores := 14;
			ELSIF (gSupS_MensajeAnom = 17)  THEN  
				Disp_SelectIndicadores := 12;
			ELSE
				Disp_SelectIndicadores := 10;			//----- Amarillo intermitente, rojo fijo. Acustico intermitente	-----//
				AccionBrazo := Anomalia_Parar;
			END_IF
			
		Identificar:
			Disp_SelectIndicadores := 1; 
	END_CASE;
END_IF;

//-------------------------------------------------------------------------------------------//
//---Envio de informacion para la funcion que gestiona anomanias en la extension del brazo---//
//-------------------------------------------------------------------------------------------//
ControlExtension(	I_TIEMPO_SEGURIDAD := T#35S,                               			//----- Tiempo de leva a recoger o extraer el brazo -----//
					I_CLEAR := gEstadoEframe=Manual OR gEstadoEframe=Automatico,
					I_RESET := (gSupS_ResetExtension OR (NOT gFinEncendido)),
					I_HABILITAR := (gEntradasAGV.Habilitar ), 
					I_DetecExtend := ((gEntradasPLC.InductivoBrazoExt OR gEntradasPLC.ParadaPrecisaBrazo) AND (gEntradasAGV.OrdenCarga OR gEntradasAGV.OrdenDescarga)) OR 
									 ((Encoder < (Encoder_Parada + 300)) AND (Encoder > (Encoder_Parada - 300)) AND gEntradasAGV.OrdenDescarga AND gEntradasAGV.OrdenDescargaB ), 
					I_DetectRecog := gEntradasPLC.InductivoBrazoRec,
					O_Estado => gDispS_ExtensionEstado);

//-------------------------------------------------------------------------------------------//
//------------Envio de informacion para la funcion que gestiona las luces y acustico---------//
//-------------------------------------------------------------------------------------------//
DISP02_Indicadores( I_SeleccionModo := Disp_SelectIndicadores,
					O_IndicadorRojo	=> gSalidasPLC.LuzRojo , 
					O_IndicadoAmarillo => gSalidasPLC.LuzAmarillo ,
					O_IndicadoVerde => gSalidasPLC.LuzVerde , 
					O_IndicadoAcustico => gSalidasPLC.Acustico);

IF (gEntradasPLC.InductivoBrazoExt OR gEntradasPLC.InductivoBrazoRec) THEN
	gSalidasPLC.Eletrofreno := FALSE;
END_IF;

//-------------------------------------------------------------------------------------------//
//----------------------------Control de la velocidad del brazo------------------------------//
//-------------------------------------------------------------------------------------------//
CASE AccionBrazo OF
	A_Extender: // Control de la velocidad en la extension del brazo em modo automatico
 		gSalidasPlc.Consigna := 0;
		gSalidasPLC.Eletrofreno := FALSE;
	
		AUX_TIMER_Extender := TRUE;
		TON_Extender( IN:=AUX_TIMER_Extender, PT:=T#1S);
	
		IF TON_Extender.Q THEN
			CASE gVelocidad OF
				E_Descargado_Tramo1:
					gSalidasPLC.Eletrofreno := TRUE; 
					gSalidasPlc.Consigna := -1500;
					gValorConsigna := gSalidasPlc.Consigna;	
				
				E_Descargado_Tramo2:
					gSalidasPLC.Eletrofreno := TRUE; 
					gSalidasPlc.Consigna := -1200; 
					gValorConsigna := gSalidasPlc.Consigna;	
					
				E_Descargado_Tramo3:
					gSalidasPLC.Eletrofreno := TRUE; 
					gSalidasPlc.Consigna := -500;
					gValorConsigna := gSalidasPlc.Consigna;	
					
				E_Cargado_Tramo1:
					gSalidasPLC.Eletrofreno := TRUE; 
					gSalidasPlc.Consigna := -800;
					gValorConsigna := gSalidasPlc.Consigna;	
					
				E_Cargado_Tramo2:
					gSalidasPLC.Eletrofreno := TRUE; 
					gSalidasPlc.Consigna := -1000;
					gValorConsigna := gSalidasPlc.Consigna;	
					
				E_Cargado_Tramo3:
					gSalidasPLC.Eletrofreno := TRUE; 
					gSalidasPlc.Consigna := -600;
					gValorConsigna := gSalidasPlc.Consigna;	
				
				SinConsigna:
					gSalidasPlc.Consigna := 0;
					gSalidasPLC.Eletrofreno := FALSE; 
					gValorConsigna := gSalidasPlc.Consigna;	
			END_CASE

			AUX_TIMER_Retraer := FALSE;
			TON_Retraer( IN:=FALSE);
		END_IF
		
	A_Recoger: // Control de la velocidad de recogida del brazo em modo automatico
		gSalidasPlc.Consigna := 0;
		gSalidasPLC.Eletrofreno := FALSE;
			
		AUX_TIMER_Retraer := TRUE;
		TON_Retraer( IN:=AUX_TIMER_Retraer, PT:=T#1S);
	
		IF TON_Retraer.Q THEN
			CASE gVelocidad OF
				R_Descargado_Tramo1:
					gSalidasPLC.Eletrofreno := TRUE; 
					gSalidasPlc.Consigna := 600;     
					gValorConsigna := gSalidasPlc.Consigna;	
					
				R_Descargado_Tramo2:
					gSalidasPLC.Eletrofreno := TRUE; 
					gSalidasPlc.Consigna := 1500;    
					gValorConsigna := gSalidasPlc.Consigna;	
					
				R_Cargado_Tramo3: 
					gSalidasPLC.Eletrofreno := TRUE; 
					gSalidasPlc.Consigna := 800;      
					gValorConsigna := gSalidasPlc.Consigna;	
					
				R_Cargado_Tramo2:
					gSalidasPLC.Eletrofreno := TRUE; 
					gSalidasPlc.Consigna := 1200;     
					gValorConsigna := gSalidasPlc.Consigna;	
					
				R_Cargado_Tramo1:
					gSalidasPLC.Eletrofreno := TRUE; 
					gSalidasPlc.Consigna := 600;  
					gValorConsigna := gSalidasPlc.Consigna;	
					
				SinConsigna:
					gSalidasPlc.Consigna := 0;
					gSalidasPLC.Eletrofreno := FALSE;
					gValorConsigna := gSalidasPlc.Consigna;	
			END_CASE

			AUX_TIMER_Extender := FALSE;
			TON_Extender( IN:=FALSE);
		END_IF
	
	A_Parar: // Parada del motor em modo automatico
		gSalidasPlc.Consigna := 0;
		gSalidasPLC.Eletrofreno := FALSE;
		
	Retener_Auto:
		gSalidasPlc.Consigna := 0;
		gSalidasPLC.Eletrofreno := FALSE;

	M_Recoger: // Recoger brazo en modo manual
		gSalidasPLC.Eletrofreno := TRUE; 
		gSalidasPlc.Consigna := SME_SPEEDRPM_MANUAL;
		
	M_Extender: // Extender brazo en modo manual
		gSalidasPLC.Eletrofreno := TRUE; 
		gSalidasPlc.Consigna := -SME_SPEEDRPM_MANUAL;
		
	M_Parar: // Parar el brazo en modo manual
		gSalidasPlc.Consigna := 0;
		gSalidasPLC.Eletrofreno := FALSE;
		
		IF gEntradasPLC.Manual_SubirLevas AND (NOT gEntradasPLC.ModoAutomatico) THEN 
			gSalidasPLC.SubirLevas := TRUE;
			gSalidasPLC.BajarLevas := FALSE;

		ELSIF gEntradasPLC.Manual_BajarLevas AND (NOT gEntradasPLC.ModoAutomatico) THEN
			gSalidasPLC.SubirLevas := FALSE;
			gSalidasPLC.BajarLevas := TRUE;
	
		ELSIF (NOT gEntradasPLC.Manual_BajarLevas) AND (NOT gEntradasPLC.Manual_SubirLevas) THEN
			gSalidasPLC.SubirLevas := FALSE;
			gSalidasPLC.BajarLevas := FALSE;
		END_IF
		
		IF gEntradasPLC.ModoAutomatico THEN
			AccionBrazo := A_Parar;
		END_IF
		
		gVelocidad := SinConsigna;
		
	Laser_Parar: // Parar el brazo despues de detectar láser
		gSalidasPlc.Consigna := 0;
	
	Setas_Parar: // Parar el brazo despues de una seta pulsada
		gSalidasPlc.Consigna := 0;

		//----- Reset de los timers -----//
		AUX_TIMER_Retraer := FALSE;
		TON_Retraer( IN:=FALSE);	
		AUX_TIMER_Extender := FALSE;
		TON_Extender( IN:=FALSE);

		
	Anomalia_Parar: // Parar el brazo despues de detectar una anomalia
		IF (gSupS_MensajeAnom <> 0) AND( gSupS_MensajeAnom <> 17) THEN
			gSalidasPlc.Consigna := 0;
			gSalidasPLC.Eletrofreno := FALSE;
			
			//----- Reset de las variables -----//
			gSalidasPLC.SubirLevas := FALSE;
			gSalidasPLC.BajarLevas := FALSE;
			gVelocidad := SinConsigna;
			AUX_CONT_Automatico := 0;
			Opt_Carga := 1;	
			Opt_Descarga := 1;
			Opt_Descarga_B := 1;
			AUX_InitSubirLevas := FALSE;
			AUX_InitBajarLevas := FALSE;
			LevasAbajoDONE := FALSE;
			LevasArribaDONE:=FALSE;
			ParadaFotocelula := FALSE;
			AUX_SubirLevas:= FALSE;
			TON_SubirLevas(IN:=FALSE);
			AUX_BajarLevas:= FALSE;
			TON_BajarLevas(IN:=FALSE);
			control_bajar:=1;
			control_subir:=1;
			AUX_EFrameDescargado := FALSE;	
			AUX_DetecionCarga := FALSE;
			TON_DetecionCarga( IN:=FALSE);
			AccionBrazo_Laser := 0;
		END_IF		
ELSE
	gSalidasPlc.Consigna := 0;
	gSalidasPLC.Eletrofreno := FALSE;
	
	gVelocidad := SinConsigna;
END_CASE

//-------------------------------------------------------------------------------------------//
//------------------------------Asignacion de anomalias del supervisor-----------------------//
//-------------------------------------------------------------------------------------------//
gSupE_AnomaliasEntrada[26] := ControlExtension.O_Anomalia.0;     //----- Anomalias que vienen de la funcion DISP01_CntrlExtensionGeneral_FB -----//
gSupE_AnomaliasEntrada[27] := ControlExtension.O_Anomalia.1;
gSupE_AnomaliasEntrada[28] := ControlExtension.O_Anomalia.2;
gSupE_AnomaliasEntrada[29] := ControlExtension.O_Anomalia.3;
gSupE_AnomaliasEntrada[30] := ControlExtension.O_Anomalia.4;
gSupE_AnomaliasEntrada[31] := ControlExtension.O_Anomalia.5;
gSupE_AnomaliasEntrada[32] := ControlExtension.O_Anomalia.6;

END_PROGRAM

// StandardPLC/Application/CÓDIGO/Seguridades/Laser_Seguridad
PROGRAM Laser_Seguridad
VAR_INPUT
	OSSD1            					:BOOL;
	OSSD2            					:BOOL;							
END_VAR							
VAR								
	SF_EQUIVALENT_LASER        			:SF_EQUIVALENT;
	SF_EMERGENCYSTOP_LASER     			:SF_EMERGENCYSTOP;
	
	NuevaRampa							:INT;
	
	EstadoCargaLaser					:OperativaARealizar;
	RangoEncoder						:BOOL;
END_VAR
VAR_OUTPUT
	AUX_Entrei							:BOOL;						
END_VAR

(*//////////////////////////////////////////////////////////////////////////////////////////////////////////////////////////////////////////////////////////////////////////////////////////////////////////////////////////////////////////////////
Laser_Seguridad (PRG)                     

Description:	Funcion de control del láser
				
///////////////////////////////////////////////////////////////////////////////////////////////////////////////////////////////////////////////////////////////////////////////////////////////////////////////////////////////////////////////////// *)

OSSD1 := gEntradasPLC.Laser_OSSD1;
OSSD2 := gEntradasPLC.Laser_OSSD2;

SF_EQUIVALENT_LASER(Activate:=1, S_CHANNELA:=OSSD1,S_CHANNELB:=OSSD2,DISCREPANCYTIME:=T#50MS);

SF_EMERGENCYSTOP_LASER(Activate:=SF_EQUIVALENT_LASER.Ready,S_ESTOPIN:=SF_EQUIVALENT_LASER.S_EquivalentOut,S_STARTRESET:=0,S_AUTORESET:=1,RESET:=0);


CASE Laser_OPT OF
	1:  // Espero que alguien se ponga en frente al laser
		IF ((NOT SF_EMERGENCYSTOP_LASER.S_ESTOPIN) AND (AccionBrazo = A_Extender) AND (NOT SetaPulsada_AUX) AND (gEstadoEframe <> Manual) AND (gEntradasAGV.OrdenCarga OR gEntradasAGV.OrdenDescarga OR (gEntradasAGV.OrdenDescarga AND gEntradasAGV.OrdenDescargaB)) ) OR
			((NOT SF_EMERGENCYSTOP_LASER.S_ESTOPIN) AND (AccionBrazo = A_Parar) AND (NOT SetaPulsada_AUX) AND (gEstadoEframe <> Manual) AND (OPT =init_cargado) AND (Opt_Descarga = 1) ) OR
			((NOT SF_EMERGENCYSTOP_LASER.S_ESTOPIN) AND (AccionBrazo = A_Parar) AND (NOT SetaPulsada_AUX) AND (gEstadoEframe <> Manual) AND (OPT =init_descargado) AND (Opt_Carga = 1) ) OR
			((NOT SF_EMERGENCYSTOP_LASER.S_ESTOPIN) AND (AccionBrazo = A_Parar) AND (NOT SetaPulsada_AUX) AND (gEstadoEframe <> Manual) AND (OPT =init_cargado_B) AND (Opt_Descarga_B = 1) ) THEN
			ParadaLaser := TRUE;
			LASER_AUX := TRUE;
			EstadoCargaLaser := OPT;
			NuevaRampa := 0;
			AUX_SalirLaser := FALSE;
			TON_SalirLaser(IN:=FALSE);
			AUX_DetecionCarga := FALSE;
			TON_DetecionCarga(IN:=FALSE);

			IF (gVelocidad = E_Cargado_Tramo1) THEN
				AccionBrazo_Laser := 1;
			ELSIF (gVelocidad = E_Cargado_Tramo2) THEN
				AccionBrazo_Laser := 2;
			ELSIF (gVelocidad = E_Cargado_Tramo3) THEN
				AccionBrazo_Laser := 3;
			ELSIF (gVelocidad = E_Descargado_Tramo1) THEN
				AccionBrazo_Laser := 4;
			ELSIF (gVelocidad = E_Descargado_Tramo2) THEN
				AccionBrazo_Laser := 5;
			ELSIF (gVelocidad = E_Descargado_Tramo3) THEN
				AccionBrazo_Laser := 6;
			ELSIF (gVelocidad = R_Cargado_Tramo1) THEN
				AccionBrazo_Laser := 7;
			ELSIF (gVelocidad = R_Cargado_Tramo2) THEN
				AccionBrazo_Laser := 8;
			ELSIF (gVelocidad = R_Cargado_Tramo3) THEN
				AccionBrazo_Laser := 9;
			ELSIF (gVelocidad = R_Descargado_Tramo1) THEN
				AccionBrazo_Laser := 10;
			ELSIF (gVelocidad = R_Descargado_Tramo2) THEN
				AccionBrazo_Laser := 11;
			END_IF

			AccionBrazo := Laser_Parar;
			gRampaVelocidad := 0;
			gSalidasPLC.Ch1_ReleSeguridad := FALSE;
			gSalidasPLC.Ch2_ReleSeguridad := FALSE;
			Laser_OPT := 2;
		END_IF
		
	2:  // Si alguien esta en frente del laser, paro el brazo
		gVelocidad := SinConsigna;		
		AUX_LaserTimer := FALSE;
		TON_Laser(IN:=FALSE);
		
		IF SF_EMERGENCYSTOP_LASER.S_ESTOPIN AND LASER_AUX THEN
			Laser_OPT := 3;
		END_IF
		
	3:  // Empiezo a contar el tiempo para el brazo empezar movimiento
		AUX_LaserTimer := TRUE;
		TON_Laser(IN:=AUX_LaserTimer,PT:=T#2S);
		
		IF TON_Laser.Q THEN
			Laser_OPT := 4;
		END_IF
		
	4:  // Empiezo movimiento del brazo
		gSalidasPLC.Ch1_ReleSeguridad := TRUE;
		gSalidasPLC.Ch2_ReleSeguridad := TRUE;

		IF ((NOT gEntradasPLC.ParadaPrecisaBrazo)  OR (NOT gEntradasPlc.InductivoBrazoExt)) AND LASER_AUX THEN
			CASE AccionBrazo_Laser OF
				1: // Velocidad de tramo 1, CARGADO EXTENDER
					gVelocidad := E_Cargado_Tramo1;

				2: // Velocidad de tramo 2, CARGADO EXTENDER
					gVelocidad := E_Cargado_Tramo2;

				3: // Velocidad de tramo 3, CARGADO EXTENDER
					gVelocidad := E_Cargado_Tramo3;

				4: // Velocidad de tramo 1, DESCARGADO EXTENDER
					gVelocidad := E_Descargado_Tramo1;

				5: // Velocidad de tramo 2, DESCARGADO EXTENDER
					gVelocidad := E_Descargado_Tramo2;

				6: // Velocidad de tramo 3, DESCARGADO EXTENDER
					gVelocidad := E_Descargado_Tramo3;

				7: // Velocidad de tramo 1, CARGADO RECOGER
					gVelocidad := R_Cargado_Tramo1;

				8: // Velocidad de tramo 2, CARGADO RECOGER
					gVelocidad := R_Cargado_Tramo2;

				9: // Velocidad de tramo 3, CARGADO RECOGER
					gVelocidad := R_Cargado_Tramo3;

				10: // Velocidad de tramo 1, DESCARGADO RECOGER
					gVelocidad := R_Descargado_Tramo1;

				11: // Velocidad de tramo 2, DESCARGADO RECOGER
					gVelocidad := R_Descargado_Tramo2;
			END_CASE	
			
			RampaCumplida := FALSE;
			AccionBrazo := A_Extender;
			LASER_AUX := FALSE;
			AUX_Entrei := TRUE;
			AUX_SalirLaser:=TRUE;
			Laser_OPT := 1;
			Reset_Consigna := TRUE;
		END_IF
END_CASE

END_PROGRAM

// StandardPLC/Application/CÓDIGO/Sub ACCIONES/ACC01_ControlManual
PROGRAM ACC01_ControlManual
VAR
	Bloqueo_Extender			:BOOL;
	Bloqueo_Recoger				:BOOL;
	
	AUX_ENTREI					:BOOL;
	Tiempo_TON_InitTeaching		:TIME;
	
	k							:INT;
END_VAR

(*//////////////////////////////////////////////////////////////////////////////////////////////////////////////////////////////////////////////////////////////////////////////////////////////////////////////////////////////////////////////////
ACC01_ControlManual (PRG)                     

Description:  Submódulo para el control manual del motor
		 
///////////////////////////////////////////////////////////////////////////////////////////////////////////////////////////////////////////////////////////////////////////////////////////////////////////////////////////////////////////////////// *)

IF LASER_AUX THEN
	gSalidasPLC.Ch1_ReleSeguridad := TRUE;
	gSalidasPLC.Ch2_ReleSeguridad := TRUE;
	LASER_AUX := FALSE;
END_IF

//-------------------------------------------------------------------------------------------//
//--------------------Reseteo de todas las variables importantes del codigo------------------//
//-------------------------------------------------------------------------------------------//
Laser := Bumper;
AUX_CONT_Automatico := 0;
OPT := indeterminado_OPT;
Opt_Carga := 1;
Opt_Carga_ANT := 0;
Opt_Descarga := 1;
Opt_Descarga_ANT := 0;
Opt_Descarga_B := 1;
Opt_DescargaB_ANT := 0;
Laser_OPT := 1;
AUX_Entrei := FALSE;
AUX_InitSubirLevas := FALSE;
AUX_InitBajarLevas := FALSE;
LevasAbajoDONE := FALSE;
LevasArribaDONE := FALSE;
ParadaFotocelula := FALSE;
AUX_SubirLevas := FALSE;
TON_SubirLevas(IN:=FALSE);
AUX_BajarLevas := FALSE;
TON_BajarLevas(IN:=FALSE);
control_bajar := 1;
control_subir := 1;
AUX_EFrameDescargado := FALSE;
AUX_DetecionCarga := FALSE;
TON_DetecionCarga(IN:=FALSE);
AccionBrazo_Laser := 0;
ACC02_ControlAutomatico.I_OrdenDescarga := FALSE;
ACC02_ControlAutomatico.I_OrdenCarga := FALSE;
ACC02_ControlAutomatico.I_OrdenDescargaB := FALSE;

//-------------------------------------------------------------------------------------------//
//------------------------------------Reseteo de anomalias-----------------------------------//
//-------------------------------------------------------------------------------------------//
FOR k := 18 TO 25 DO
	gSupE_AnomaliasEntrada[k] := 1;
END_FOR

gSupE_AnomaliasEntrada[32] := 1;
gSupE_AnomaliasEntrada[33] := 1;
gSupE_AnomaliasEntrada[35] := 1;

//-------------------------------------------------------------------------------------------//
//---------------------------------------Control Manual--------------------------------------//
//-------------------------------------------------------------------------------------------//
IF (gEntradasPlc.InductivoBrazoExt AND (NOT gEntradasPlc.InductivoBrazoRec)) THEN
	Bloqueo_Extender := TRUE;
	Bloqueo_Recoger := FALSE;
ELSIF (gEntradasPlc.InductivoBrazoRec AND (NOT gEntradasPlc.InductivoBrazoExt)) THEN
	Bloqueo_Extender := FALSE;
	Bloqueo_Recoger := TRUE;
ELSIF ((NOT gEntradasPlc.InductivoBrazoRec) AND (NOT gEntradasPlc.InductivoBrazoExt)) THEN
	Bloqueo_Extender := FALSE;
	Bloqueo_Recoger := FALSE;
	PararMotorManual := FALSE;
END_IF
	
IF gEntradasPLC.Manual_RecogerBrazo AND (NOT Bloqueo_Recoger) THEN
	AccionBrazo := M_Recoger;

	IF (gEntradasPlc.InductivoBrazoRec AND (NOT gEntradasPlc.InductivoBrazoExt) ) THEN
		AccionBrazo := M_Parar;
	END_IF

ELSIF gEntradasPLC.Manual_ExtenderBrazo AND (NOT Bloqueo_Extender) THEN 
	AccionBrazo := M_Extender;
	AUX_ENTREI := TRUE;
	IF (gEntradasPlc.InductivoBrazoExt AND (NOT gEntradasPlc.InductivoBrazoRec)) THEN
		AccionBrazo := M_Parar;
	END_IF

ELSIF (NOT gEntradasPLC.Manual_ExtenderBrazo) OR (NOT gEntradasPLC.Manual_RecogerBrazo) THEN
	AccionBrazo := M_Parar;	
END_IF

IF gEntradasPlc.InductivoBrazoRec AND (AccionBrazo = M_Parar) AND (NOT gEntradasPLC.ModoAutomatico) THEN
	TON_InitTeaching(IN:=gEntradasPLC.BotonRearme, PT:=T#500MS, ET => Tiempo_TON_InitTeaching);
	
	IF TON_InitTeaching.Q THEN
		DISP03_EncoderTeaching();
	END_IF
END_IF

IF gEntradasPlc.InductivoBrazoExt AND (AccionBrazo = M_Parar) AND (NOT gEntradasPLC.ModoAutomatico) THEN
	TON_InitTeaching(IN:=gEntradasPLC.BotonRearme, PT:=T#500MS, ET => Tiempo_TON_InitTeaching);
	
	IF TON_InitTeaching.Q THEN
		DISP03_EncoderTeaching();
	END_IF
END_IF

IF (NOT gEntradasPlc.InductivoBrazoExt) AND (NOT gEntradasPlc.InductivoBrazoRec) AND (AccionBrazo = M_Parar) AND (Encoder < TeachingOperativaB) AND (NOT gEntradasPLC.ModoAutomatico) THEN
	TON_InitTeaching(IN:=gEntradasPLC.BotonRearme, PT:=T#500MS, ET => Tiempo_TON_InitTeaching);
	
	IF TON_InitTeaching.Q THEN
		DISP03_EncoderTeaching();
	END_IF
END_IF

END_PROGRAM

// StandardPLC/Application/CÓDIGO/Sub Dispositivos/DISP03_EncoderTeaching
PROGRAM DISP03_EncoderTeaching
VAR
	TON_Encoder						:TON;
	TON_Encoder_OFF					:TON;
	Tempo_Actual_Encoder 			:TIME;
	Tempo_Actual_Encoder_OFF 		:TIME;
END_VAR

(*//////////////////////////////////////////////////////////////////////////////////////////////////////////////////////////////////////////////////////////////////////////////////////////////////////////////////////////////////////////////////
DISP03_EncoderTeaching (PRG)                     

Description:	Bloque de control del modo teaching del encoder
				 
///////////////////////////////////////////////////////////////////////////////////////////////////////////////////////////////////////////////////////////////////////////////////////////////////////////////////////////////////////////////////// *)

CASE gTeachingEncoder OF
	1:  // Miramos si tenemos el E-Frame en modo manual y la accion del brazo como parado
		IF (NOT gEntradasPLC.ModoAutomatico) AND (AccionBrazo = M_Parar) THEN
			StartCount_Encoder := TRUE;
			gTeachingEncoder := 2;
		END_IF
		
	2: // Miramos si el utilizador pulsa el boton rearme durante 8 segundos y iniciamos el timer
		TON_Encoder( IN:=(StartCount_Encoder AND gEntradasPLC.BotonRearme), PT:=T#8S, ET => Tempo_Actual_Encoder );
		
		IF TON_Encoder.Q THEN
			gTeachingEncoder := 3;
		END_IF
		
	3: // Guardamos el valor del encoder en la variable persistente
		IF gEntradasPlc.InductivoBrazoRec THEN
			gEncoder_Absoluto := Encoder;
			PARAMETRIZACION();
			TeachingDone := TRUE;
			gTeachingEncoder := 4;
			
		ELSIF gEntradasPlc.InductivoBrazoExt THEN
			gEncoder_AbsolutoExtendido := Encoder;
			PARAMETRIZACION();
			TeachingDone := TRUE;
			gTeachingEncoder := 4;
			
		ELSIF (NOT gEntradasPlc.InductivoBrazoRec) AND (NOT gEntradasPlc.InductivoBrazoExt) THEN
			gEncoder_OperativaB := Encoder;
			PARAMETRIZACION();
			TeachingDone := TRUE;
			gTeachingEncoder := 4;
			
		END_IF
		
	4: // Iniciamos el timer de 1 s para apagar la baliza y buzzer
		TON_Encoder_OFF( IN:=TeachingDone, PT:=T#1S, ET => Tempo_Actual_Encoder_OFF );
		
		IF TON_Encoder_OFF.Q THEN
			gTeachingEncoder := 5;
		END_IF
	
	5: // Reseteamos los timers y las variables utilizadas anteriormente
		TeachingDone := FALSE;
		StartCount_Encoder := FALSE;
		
		TON_Encoder(IN:=FALSE);
		TON_Encoder_OFF(IN:=FALSE);
		TON_InitTeaching(IN:=FALSE);
		
		gTeachingEncoder := 1;
END_CASE

END_PROGRAM

// StandardPLC/Application/CÓDIGO/Sub ACCIONES/ACC00_SalidasDesactivadas
PROGRAM ACC00_SalidasDesactivadas
VAR
END_VAR

(*//////////////////////////////////////////////////////////////////////////////////////////////////////////////////////////////////////////////////////////////////////////////////////////////////////////////////////////////////////////////////
ACC00_SalidasDesactivadas (PRG)                     

Description:	Submódulo para la desactivación de las salidas del E-Frame
				Lo utilizamos para el modo degradado
				
///////////////////////////////////////////////////////////////////////////////////////////////////////////////////////////////////////////////////////////////////////////////////////////////////////////////////////////////////////////////////// *)

//-------------------------------------------------------------------------------------------//
//---------------------------Desactivacion del motor de las levas----------------------------//
//-------------------------------------------------------------------------------------------//
gSalidasPLC.SubirLevas := FALSE;
gSalidasPLC.BajarLevas := FALSE;

